(* Kommunikation mit der KL6581. *)
(* Communication with the KL6581. *)
fbKL6581(
	bInit			:= bInitCom,
	nIdx			:= 2,
	stKL6581_in		:= stKL6581_In,
	stKL6581_out	:= stKL6581_Out,
	bReady			=> ,
	bBusy			=> ,
	bError			=> ,
	iErrorID		=> ,
	str_KL6581		=> stKL6581);

GVL_AHDataModbus.EnOceanError	:= TO_UINT(fbKL6581.iErrorID);
(* Warten bis der Kommunikationsbaustein initialisiert wurde.*)
(* Wait until the communication function block has been initialized. *)
IF (NOT fbKL6581.bReady) THEN
	RETURN;
END_IF

FOR nSearchIdx:= 1 TO 8 DO
	arrEnOcean_Search[nSearchIdx](
		bStart:= TRUE, 
		str_KL6581:= stKL6581 , 
		byNode:= nSearchIdx, 
		bReceive=> , 
		iDevices=>arrDevices[nSearchIdx] , 
		ar_ID=> );
		
		MEMCPY(ADR(arrID[nSearchIdx,0]), ADR(arrEnOcean_Search[nSearchIdx].ar_ID), SIZEOF(arrEnOcean_Search[nSearchIdx].ar_ID)); 
END_FOR

//A_Gang_3_364()

A_Rum_2_351();
A_Rum_2_352();
A_Rum_2_353();
A_Rum_2_354();
A_Rum_2_355();
A_Rum_2_356();
A_Rum_2_357();
A_Rum_3_365();
A_Rum_3_361();
A_Rum_3_366();
A_Rum_3_367();
A_Rum_3_368();
A_Rum_3_369();
A_Rum_3_370();
//AtriumNiveau
A_AtriumNiveau();

ACTION A_AtriumNiveau:
fbAtriumNiveau_Tryk_PladeB(
	str_KL6581:=stKL6581 , 
	byNode:=0, 
	dw_ID:= 16#0029B92D, 
	str_EnOceanSwitch=> GVL_EnOcean.strEnOceanSwitch_AtriumNiveau_PladeB,
	by_Node=> , 
	bReceive=> );
(*
fbAtriumNiveau_Tryk_Sevice(
	str_KL6581:=stKL6581 , 
	byNode:=0, 
	dw_ID:= 16#00FEE4FE87, 
	str_EnOceanSwitch=> GVL_EnOcean.strEnOceanSwitch_AtriumNiveau_Service, 
	by_Node=> , 
	bReceive=> );
*)
END_ACTION

ACTION A_Rum_2_351:
fbRum_2_351_Tryk(
	str_KL6581:=stKL6581 , 
	byNode:=byNode_2 , 
	dw_ID:= 16#290EEB, 
	str_EnOceanSwitch=> GVL_EnOcean.strEnOceanSwitch_Rum_2_351, 
	by_Node=> , 
	bReceive=> );
END_ACTION

ACTION A_Rum_2_352:
fbRum_2_352_Tryk(
	str_KL6581:=stKL6581 , 
	byNode:=byNode_2 , 
	dw_ID:= 16#2F3276, 
	str_EnOceanSwitch=> GVL_EnOcean.strEnOceanSwitch_Rum_2_352, 
	by_Node=> , 
	bReceive=> );
END_ACTION

ACTION A_Rum_2_353:
fbRum_2_353_Tryk(
	str_KL6581:=stKL6581 , 
	byNode:=byNode_2 , 
	dw_ID:= 16#002E7C1F, 
	str_EnOceanSwitch=> GVL_EnOcean.strEnOceanSwitch_Rum_2_353, 
	by_Node=> , 
	bReceive=> );
END_ACTION

ACTION A_Rum_2_354:
fbRum_2_354_Tryk(
	str_KL6581:=stKL6581 , 
	byNode:=byNode_2 , 
	dw_ID:= 16#002F6627, 
	str_EnOceanSwitch=> GVL_EnOcean.strEnOceanSwitch_Rum_2_354, 
	by_Node=> , 
	bReceive=> );
END_ACTION

ACTION A_Rum_2_355:
fbRum_2_355_Tryk(
	str_KL6581:=stKL6581 , 
	byNode:=byNode_2 , 
	dw_ID:= 16#0029AD66, 
	str_EnOceanSwitch=> GVL_EnOcean.strEnOceanSwitch_Rum_2_355, 
	by_Node=> , 
	bReceive=> );
END_ACTION

ACTION A_Rum_2_356:
fbRum_2_356_Tryk(
	str_KL6581:=stKL6581 , 
	byNode:=byNode_2 , 
	dw_ID:= 16#0029AD36, 
	str_EnOceanSwitch=> GVL_EnOcean.strEnOceanSwitch_Rum_2_356, 
	by_Node=> , 
	bReceive=> );
END_ACTION

ACTION A_Rum_2_357:
fbRum_2_357_Tryk(
	str_KL6581:=stKL6581 , 
	byNode:=byNode_2 , 
	dw_ID:= 16#0029AD42, 
	str_EnOceanSwitch=> GVL_EnOcean.strEnOceanSwitch_Rum_2_357, 
	by_Node=> , 
	bReceive=> );
END_ACTION

ACTION A_Rum_3_361:
fbRum_3_361_Tryk_1(
	str_KL6581:=stKL6581 , 
	byNode:=byNode_2 , 
	dw_ID:= 16#29AD02, 
	str_EnOceanSwitch=> GVL_EnOcean.strEnOceanSwitch_Rum_3_361_1, 
	by_Node=> , 
	bReceive=> );


fbRum_3_361_Tryk_2(
	str_KL6581:=stKL6581 , 
	byNode:=byNode_2 , 
	dw_ID:= 16#0029ACFE, 
	str_EnOceanSwitch=> GVL_EnOcean.strEnOceanSwitch_Rum_3_361_2, 
	by_Node=> , 
	bReceive=> );
END_ACTION

ACTION A_Rum_3_365:
fbRum_3_365_Tryk(
	str_KL6581:=stKL6581 , 
	byNode:=byNode_2 , 
	dw_ID:= 16#0029AD2C, 
	str_EnOceanSwitch=> GVL_EnOcean.strEnOceanSwitch_Rum_3_365, 
	by_Node=> , 
	bReceive=> );
END_ACTION

ACTION A_Rum_3_366:
fbRum_3_366_Tryk(
	str_KL6581:=stKL6581 , 
	byNode:=byNode_2 , 
	dw_ID:= 16#0029AD33, 
	str_EnOceanSwitch=> GVL_EnOcean.strEnOceanSwitch_Rum_3_366, 
	by_Node=> , 
	bReceive=> );
END_ACTION

ACTION A_Rum_3_367:
fbRum_3_367_Tryk(
	str_KL6581:=stKL6581 , 
	byNode:=byNode_2 , 
	dw_ID:= 16#0029AD1B, 
	str_EnOceanSwitch=> GVL_EnOcean.strEnOceanSwitch_Rum_3_367, 
	by_Node=> , 
	bReceive=> );
END_ACTION

ACTION A_Rum_3_368:
fbRum_3_368_Tryk(
	str_KL6581:=stKL6581 , 
	byNode:=byNode_2 , 
	dw_ID:= 16#0029AD61, 
	str_EnOceanSwitch=> GVL_EnOcean.strEnOceanSwitch_Rum_3_368, 
	by_Node=> , 
	bReceive=> );
END_ACTION

ACTION A_Rum_3_369:
fbRum_3_369_Tryk(
	str_KL6581:=stKL6581 , 
	byNode:=byNode_2 , 
	dw_ID:= 16#0029AD37, 
	str_EnOceanSwitch=> GVL_EnOcean.strEnOceanSwitch_Rum_3_369, 
	by_Node=> , 
	bReceive=> );
END_ACTION

ACTION A_Rum_3_370:
fbRum_3_370_Tryk(
	str_KL6581:=stKL6581 , 
	byNode:=byNode_2 , 
	dw_ID:= 16#002F665E, 
	str_EnOceanSwitch=> GVL_EnOcean.strEnOceanSwitch_Rum_3_370, 
	by_Node=> , 
	bReceive=> );
END_ACTION

END_PROGRAM

// ---- POUs/MAIN.TcPOU
PROGRAM MAIN
VAR
	nAlive: INT;
	breset: BOOL;
	nDemoVariable : INT;
	nCX8200_State	AT %I*	: UINT;
END_VAR

VAR PERSISTENT
	nDemoVar_Persist: INT;
END_VAR

nAlive:= nAlive + 1;
GVL_AHDataModbus.nCX8200_State_MB := nCX8200_State;

P_SystemDK.M_nCyclic(bReset := breset );
P_DALI_DIAG();
//P_EnOcean(); Testing fast task
DALI_Commissioning();
P_DALI_Energy_Line();
P_AHModbusComm();
P_Foldedoer_3_366();

//Gange
P_Gang_2_350();
P_Gang_3_362A();
P_Gang_3_363A();
P_Gang_3_363B();
P_Gang_3_364();
P_gang_3_309();
//Rum
P_Rum_2_351();
P_Rum_2_352();
P_Rum_2_353();
P_Rum_2_354();
P_Rum_2_355();
P_Rum_2_356();
P_Rum_2_357();
P_Rum_3_361();
P_Rum_3_366();
P_Rum_3_367();
P_Rum_3_368();
P_Rum_3_369();
P_Rum_3_370();

//P_Lys_Grp0();
//P_DALI_Energy_Firmware_Test();
P_Trappe();

END_PROGRAM

// ---- POUs/Tester/P_Test_TypeA.TcPOU
PROGRAM P_Test_TypeA
VAR
	fbTA: FB_FunctionType_A;
	bButtonZone1 			: BOOL;
	bButtonZone2 			: BOOL;
	bPIR 					: BOOL;
	fLuxOn 					: REAL := 500;
	fLuxDim 				: REAL := 200;
	tPIRDim 				: TIME := T#15M;
	tPIROff 				: TIME := T#30M;
	
	//Output from FB
	fLuxZone1 				: REAL;
	bDimUp					: BOOL:= FALSE;
	bDimDwn 				: BOOL:= FALSE;
	bOnZone1 				: BOOL;
	bOffZone1 				: BOOL:= TRUE;
	bAutoZone1 				: BOOL:= TRUE;
	
	bAutoZone2 				: BOOL:= TRUE;
	bOnZone2 				: BOOL;
	bOffZone2 				: BOOL:= TRUE;
	
END_VAR


fbTA(
	bButtonZone1:= bButtonZone1, 
	bButtonZone2:= bButtonZone2 , 
	bPIR:= bPIR, 
	fLuxOn:= fLuxOn, 
	fLuxDim:= fLuxDim, 
	tPIRDim:= tPIRDim, 
	tPIROff:= tPIROff, 
	fLuxZone1=> fLuxZone1, 
	bDimUp=> bDimUp , 
	bDimDwn=> bDimDwn, 
	bOnZone1=> bOnZone1, 
	bOffZone1=> bOffZone1, 
	bAutoZone1=> bAutoZone1, 
	bAutoZone2=> bAutoZone2, 
	bOnZone2=> bOnZone2, 
	bOffZone2=> bOffZone2);

END_PROGRAM

// ---- GlobalTextList.TcGTLO
TEXTLIST GlobalTextList
  621 = '%d'
  6 = 'Bottom Button'
  482 = 'Button 1'
  720 = 'Button 2'
  1902 = 'DALI Line:'
  1180 = 'DI1 falling edge'
  1218 = 'DI1 rising edge'
  1726 = 'DI2 falling edge'
  1876 = 'DI2 rising edge'
  519 = 'Dim Dwn'
  63 = 'Dim Up'
  2135 = 'Do not lock process image in case of \nDALI commands from DI1 or DI2'
  967 = 'Gang 1.312A'
  256 = 'Gang 1.315'
  906 = 'Gang 1.316'
  207 = 'Gang 2.344'
  66 = 'Gang 2.344A'
  583 = 'Gang 2.350'
  985 = 'Gang 3.362A'
  67 = 'Gang 3.363A'
  173 = 'Gang 3.363B'
  406 = 'Gang 4.308'
  524 = 'Gang 6.310'
  316 = 'Gang 7.301'
  492 = 'Internal DALI power supply disabled'
  1771 = 'K-Bus Watchdog'
  1811 = 'Lockable bytes: changeable if "Offset 2" has the Value 85 (0x55).\nFor changing use decimal value.'
  43 = 'Lys Auto'
  444 = 'Lys Rum'
  489 = 'Lys Zone 1'
  2046 = 'Memory Bank:'
  23 = 'Name'
  926 = 'Name of byte in memory bank'
  22 = 'Offset'
  1329 = 'Offset in memory bank'
  708 = 'PIR'
  457 = 'PIR status'
  373 = 'Read'
  2418 = 'Reset inactive process image'
  874 = 'Rum 1.106'
  65 = 'Rum 1.108'
  175 = 'Rum 1.111A'
  924 = 'Rum 1.111C'
  219 = 'Rum 1.111D'
  690 = 'Rum 1.111E'
  912 = 'Rum 1.115'
  126 = 'Rum 1.118'
  215 = 'Rum 1.312A'
  725 = 'Rum 1.318'
  839 = 'Rum 1.319'
  456 = 'Rum 1.320'
  800 = 'Rum 1.321'
  622 = 'Rum 1.322'
  646 = 'Rum 1.323'
  966 = 'Rum 1.324'
  95 = 'Rum 1.325'
  335 = 'Rum 1.326'
  150 = 'Rum 1.327'
  651 = 'Rum 1.328'
  980 = 'Rum 1.330'
  262 = 'Rum 1115'
  642 = 'Rum 2.341'
  978 = 'Rum 2.345'
  736 = 'Rum 2.349'
  593 = 'Rum 2.351'
  122 = 'Rum 2.352'
  27 = 'Rum 2.353'
  41 = 'Rum 2.354'
  697 = 'Rum 2.355'
  826 = 'Rum 2.356'
  561 = 'Rum 2.357'
  415 = 'Rum 3.365'
  981 = 'Rum 3.366'
  865 = 'Rum 3.367'
  212 = 'Rum 3.368'
  921 = 'Rum 3.369'
  329 = 'Rum 3.370'
  430 = 'Rum 6.310 Sofagruppe'
  348 = 'Rum 6.327'
  891 = 'Rum 6.328'
  11 = 'Rum 6.329'
  72 = 'Rum 6.330B'
  197 = 'Rum 6.331'
  564 = 'Rum 6.333'
  997 = 'Rum 6.337'
  31 = 'Rum 6_330A'
  1041 = 'Short Address:'
  395 = 'SP_Lux: %.0f'
  525 = 'SP_Lux: %f'
  2458 = 'Terminal Event'
  849 = 'Test Type A'
  973 = 'Top Button'
  24 = 'Value Dec'
  1435 = 'Value decimal'
  25 = 'Value Hex'
  2231 = 'Value hexadecimal,\nto change use\nvalue decimal'
  374 = 'Write'
  1047 = 'Write default values'
  490 = 'Write parameters'
END_TEXTLIST

// ---- POUs/Alle_Rum/Gange/Gang_3_362A/Visualization_3_362A.TcVIS
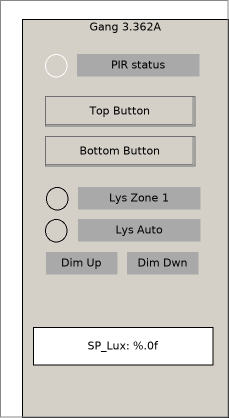
VISUALIZATION Visualization_3_362A  // 229x418
    RoundedRectangle (22,19 207x399), "Gang 3.362A"
    Rectangle (33,327 180x38), "SP_Lux: %.0f", text variable: P_Gang_3_362A.fbLys.fbLightCtrl.fLuxZone1
    Button (45,96 150x30), "Top Button"
        tap P_Gang_3_362A.bTopButtonZone1_Visu
    Button (45,136 150x30), "Bottom Button"
        tap P_Gang_3_362A.bBottomButtonZone1_Visu
    Ellipse (46,187 22x23), colour toggle: P_Gang_3_362A.fbLys.fbLightCtrl.bOnZone1
    Rectangle (78,187 122x22), "Lys Zone 1"
    Rectangle (46,252 71x22), "Dim Up", colour toggle: P_Gang_3_362A.fbLys.fbLightCtrl.bDimUp
    Rectangle (127,252 71x22), "Dim Dwn", colour toggle: P_Gang_3_362A.fbLys.fbLightCtrl.bDimDwn
    Ellipse (45,219 22x23), colour toggle: P_Gang_3_362A.fbLys.fbLightCtrl.bAutoZone1
    Rectangle (78,219 122x22), "Lys Auto"
    Ellipse (45,54 22x23), colour toggle: P_Gang_3_362A.fbLys.fbLightCtrl.bPIR
    Rectangle (77,54 122x22), "PIR status"
END_VISUALIZATION

// ---- POUs/Alle_Rum/Gange/Gang_3_363A/Visualization_3_363A.TcVIS
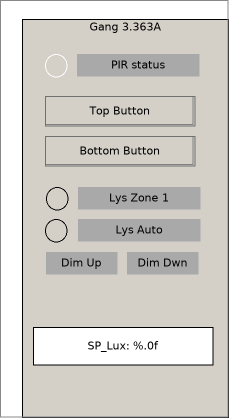
VISUALIZATION Visualization_3_363A  // 229x418
    RoundedRectangle (22,19 207x399), "Gang 3.363A"
    Rectangle (33,327 180x38), "SP_Lux: %.0f", text variable: P_Gang_3_363A.fbLys.fbLightCtrl.fLuxZone1
    Button (45,96 150x30), "Top Button"
        tap P_Gang_3_363A.bTopButtonZone1_Visu
    Button (45,136 150x30), "Bottom Button"
        tap P_Gang_3_363A.bBottomButtonZone1_Visu
    Ellipse (46,187 22x23), colour toggle: P_Gang_3_363A.fbLys.fbLightCtrl.bOnZone1
    Rectangle (78,187 122x22), "Lys Zone 1"
    Rectangle (46,252 71x22), "Dim Up", colour toggle: P_Gang_3_363A.fbLys.fbLightCtrl.bDimUp
    Rectangle (127,252 71x22), "Dim Dwn", colour toggle: P_Gang_3_363A.fbLys.fbLightCtrl.bDimDwn
    Ellipse (45,219 22x23), colour toggle: P_Gang_3_363A.fbLys.fbLightCtrl.bAutoZone1
    Rectangle (78,219 122x22), "Lys Auto"
    Ellipse (45,54 22x23), colour toggle: P_Gang_3_363A.fbLys.fbLightCtrl.bPIR
    Rectangle (77,54 122x22), "PIR status"
END_VISUALIZATION

// ---- POUs/Alle_Rum/Gange/Gang_3_363B/Visualization_3_363B.TcVIS
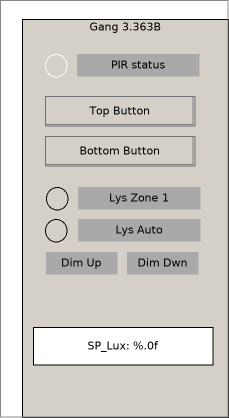
VISUALIZATION Visualization_3_363B  // 229x418
    RoundedRectangle (22,19 207x399), "Gang 3.363B"
    Rectangle (33,327 180x38), "SP_Lux: %.0f", text variable: P_Gang_3_362A.fbLys.fbLightCtrl.fLuxZone1
    Button (45,96 150x30), "Top Button"
        tap P_Gang_3_363B.bTopButtonZone1_Visu
    Button (45,136 150x30), "Bottom Button"
        tap P_Gang_3_363B.bBottomButtonZone1_Visu
    Ellipse (46,187 22x23), colour toggle: P_Gang_3_363B.fbLys.fbLightCtrl.bOnZone1
    Rectangle (78,187 122x22), "Lys Zone 1"
    Rectangle (46,252 71x22), "Dim Up", colour toggle: P_Gang_3_363B.fbLys.fbLightCtrl.bDimUp
    Rectangle (127,252 71x22), "Dim Dwn", colour toggle: P_Gang_3_363B.fbLys.fbLightCtrl.bDimDwn
    Ellipse (45,219 22x23), colour toggle: P_Gang_3_363B.fbLys.fbLightCtrl.bAutoZone1
    Rectangle (78,219 122x22), "Lys Auto"
    Ellipse (45,54 22x23), colour toggle: P_Gang_3_363B.fbLys.fbLightCtrl.bPIR
    Rectangle (77,54 122x22), "PIR status"
END_VISUALIZATION

// ---- POUs/Alle_Rum/Gange/Gang_3_364/Visualization_3_364.TcVIS
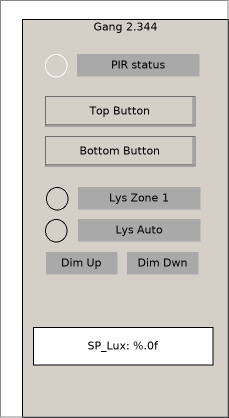
VISUALIZATION Visualization_3_364  // 229x418
    RoundedRectangle (22,19 207x399), "Gang 2.344"
    Rectangle (33,327 180x38), "SP_Lux: %.0f", text variable: P_Gang_3_364.fbLys.fbLightCtrl.fLuxZone1
    Button (45,96 150x30), "Top Button"
        tap P_Gang_3_364.bTopButtonZone1_Visu
    Button (45,136 150x30), "Bottom Button"
        tap P_Gang_3_364.bBottomButtonZone1_Visu
    Ellipse (46,187 22x23), colour toggle: P_Gang_3_364.fbLys.fbLightCtrl.bOnZone1
    Rectangle (78,187 122x22), "Lys Zone 1"
    Rectangle (46,252 71x22), "Dim Up", colour toggle: P_Gang_3_364.fbLys.fbLightCtrl.bDimUp
    Rectangle (127,252 71x22), "Dim Dwn", colour toggle: P_Gang_3_364.fbLys.fbLightCtrl.bDimDwn
    Ellipse (45,219 22x23), colour toggle: P_Gang_3_364.fbLys.fbLightCtrl.bAutoZone1
    Rectangle (78,219 122x22), "Lys Auto"
    Ellipse (45,54 22x23), colour toggle: P_Gang_3_364.fbLys.fbLightCtrl.bPIR
    Rectangle (77,54 122x22), "PIR status"
END_VISUALIZATION

// ---- POUs/Alle_Rum/Gange/Gang_2_350/Visualization_2_350.TcVIS
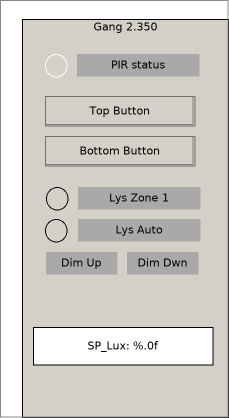
VISUALIZATION Visualization_2_350  // 229x418
    RoundedRectangle (22,19 207x399), "Gang 2.350"
    Rectangle (33,327 180x38), "SP_Lux: %.0f", text variable: P_Gang_3_364.fbLys.fbLightCtrl.fLuxZone1
    Button (45,96 150x30), "Top Button"
        tap P_Gang_2_350.bTopButtonZone1_Visu
    Button (45,136 150x30), "Bottom Button"
        tap P_Gang_2_350.bBottomButtonZone1_Visu
    Ellipse (46,187 22x23), colour toggle: P_Gang_2_350.fbLys.fbLightCtrl.bOnZone1
    Rectangle (78,187 122x22), "Lys Zone 1"
    Rectangle (46,252 71x22), "Dim Up", colour toggle: P_Gang_2_350.fbLys.fbLightCtrl.bDimUp
    Rectangle (127,252 71x22), "Dim Dwn", colour toggle: P_Gang_2_350.fbLys.fbLightCtrl.bDimDwn
    Ellipse (45,219 22x23), colour toggle: P_Gang_2_350.fbLys.fbLightCtrl.bAutoZone1
    Rectangle (78,219 122x22), "Lys Auto"
    Ellipse (45,54 22x23), colour toggle: P_Gang_2_350.fbLys.fbLightCtrl.bPIR
    Rectangle (77,54 122x22), "PIR status"
END_VISUALIZATION

// ---- POUs/Alle_Rum/Rum_Med_DALI_Pir/Rum_2_351/Visualization_2_351.TcVIS
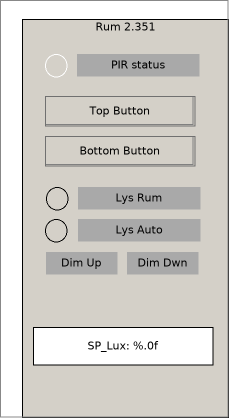
VISUALIZATION Visualization_2_351  // 229x418
    RoundedRectangle (22,19 207x399), "Rum 2.351"
    Rectangle (33,327 180x38), "SP_Lux: %.0f", text variable: P_Rum_2_351.fbLys.fbLightCtrl.fLuxZone1
    Button (45,96 150x30), "Top Button"
        tap P_Rum_2_351.bTopButtonZone1_Visu
    Button (45,136 150x30), "Bottom Button"
        tap P_Rum_2_351.bBottomButtonZone1_Visu
    Ellipse (46,187 22x23), colour toggle: P_Rum_2_351.fbLys.fbLightCtrl.bOnZone1
    Rectangle (78,187 122x22), "Lys Rum"
    Rectangle (46,252 71x22), "Dim Up", colour toggle: P_Rum_2_351.fbLys.fbLightCtrl.bDimUp
    Rectangle (127,252 71x22), "Dim Dwn", colour toggle: P_Rum_2_351.fbLys.fbLightCtrl.bDimDwn
    Ellipse (45,219 22x23), colour toggle: P_Rum_2_351.fbLys.fbLightCtrl.bAutoZone1
    Rectangle (78,219 122x22), "Lys Auto"
    Ellipse (45,54 22x23), colour toggle: P_Rum_2_351.fbLys.fbLightCtrl.bPIR
    Rectangle (77,54 122x22), "PIR status"
END_VISUALIZATION

// ---- POUs/Alle_Rum/Rum_Med_DALI_Pir/Rum_2_352/Visualization_2_352.TcVIS
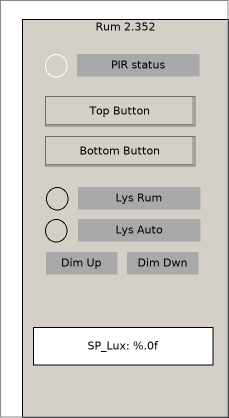
VISUALIZATION Visualization_2_352  // 229x418
    RoundedRectangle (22,19 207x399), "Rum 2.352"
    Rectangle (33,327 180x38), "SP_Lux: %.0f", text variable: P_Rum_2_351.fbLys.fbLightCtrl.fLuxZone1
    Button (45,96 150x30), "Top Button"
        tap P_Rum_2_352.bTopButtonZone1_Visu
    Button (45,136 150x30), "Bottom Button"
        tap P_Rum_2_352.bBottomButtonZone1_Visu
    Ellipse (46,187 22x23), colour toggle: P_Rum_2_352.fbLys.fbLightCtrl.bOnZone1
    Rectangle (78,187 122x22), "Lys Rum"
    Rectangle (46,252 71x22), "Dim Up", colour toggle: P_Rum_2_352.fbLys.fbLightCtrl.bDimUp
    Rectangle (127,252 71x22), "Dim Dwn", colour toggle: P_Rum_2_352.fbLys.fbLightCtrl.bDimDwn
    Ellipse (45,219 22x23), colour toggle: P_Rum_2_352.fbLys.fbLightCtrl.bAutoZone1
    Rectangle (78,219 122x22), "Lys Auto"
    Ellipse (45,54 22x23), colour toggle: P_Rum_2_352.fbLys.fbLightCtrl.bPIR
    Rectangle (77,54 122x22), "PIR status"
END_VISUALIZATION

// ---- POUs/Alle_Rum/Rum_Med_DALI_Pir/Rum_2_353/Visualization_2_353.TcVIS
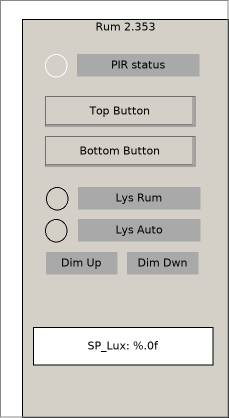
VISUALIZATION Visualization_2_353  // 229x418
    RoundedRectangle (22,19 207x399), "Rum 2.353"
    Rectangle (33,327 180x38), "SP_Lux: %.0f", text variable: P_Rum_2_353.fbLys.fbLightCtrl.fLuxZone1
    Button (45,96 150x30), "Top Button"
        tap P_Rum_2_353.bTopButtonZone1_Visu
    Button (45,136 150x30), "Bottom Button"
        tap P_Rum_2_353.bBottomButtonZone1_Visu
    Ellipse (46,187 22x23), colour toggle: P_Rum_2_353.fbLys.fbLightCtrl.bOnZone1
    Rectangle (78,187 122x22), "Lys Rum"
    Rectangle (46,252 71x22), "Dim Up", colour toggle: P_Rum_2_353.fbLys.fbLightCtrl.bDimUp
    Rectangle (127,252 71x22), "Dim Dwn", colour toggle: P_Rum_2_353.fbLys.fbLightCtrl.bDimDwn
    Ellipse (45,219 22x23), colour toggle: P_Rum_2_353.fbLys.fbLightCtrl.bAutoZone1
    Rectangle (78,219 122x22), "Lys Auto"
    Ellipse (45,54 22x23), colour toggle: P_Rum_2_353.fbLys.fbLightCtrl.bPIR
    Rectangle (77,54 122x22), "PIR status"
END_VISUALIZATION

// ---- POUs/Alle_Rum/Rum_Med_DALI_Pir/Rum_2_354/Visualization_2_354.TcVIS
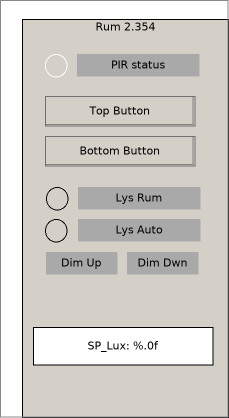
VISUALIZATION Visualization_2_354  // 229x418
    RoundedRectangle (22,19 207x399), "Rum 2.354"
    Rectangle (33,327 180x38), "SP_Lux: %.0f", text variable: P_Rum_2_354.fbLys.fbLightCtrl.fLuxZone1
    Button (45,96 150x30), "Top Button"
        tap P_Rum_2_354.bTopButtonZone1_Visu
    Button (45,136 150x30), "Bottom Button"
        tap P_Rum_2_354.bBottomButtonZone1_Visu
    Ellipse (46,187 22x23), colour toggle: P_Rum_2_354.fbLys.fbLightCtrl.bOnZone1
    Rectangle (78,187 122x22), "Lys Rum"
    Rectangle (46,252 71x22), "Dim Up", colour toggle: P_Rum_2_354.fbLys.fbLightCtrl.bDimUp
    Rectangle (127,252 71x22), "Dim Dwn", colour toggle: P_Rum_2_354.fbLys.fbLightCtrl.bDimDwn
    Ellipse (45,219 22x23), colour toggle: P_Rum_2_354.fbLys.fbLightCtrl.bAutoZone1
    Rectangle (78,219 122x22), "Lys Auto"
    Ellipse (45,54 22x23), colour toggle: P_Rum_2_354.fbLys.fbLightCtrl.bPIR
    Rectangle (77,54 122x22), "PIR status"
END_VISUALIZATION

// ---- POUs/Alle_Rum/Rum_Med_DALI_Pir/Rum_2_357/Visualization_2_357.TcVIS
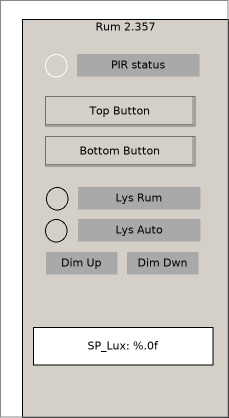
VISUALIZATION Visualization_2_357  // 229x418
    RoundedRectangle (22,19 207x399), "Rum 2.357"
    Rectangle (33,327 180x38), "SP_Lux: %.0f", text variable: P_Rum_2_357.fbLys.fbLightCtrl.fLuxZone1
    Button (45,96 150x30), "Top Button"
        tap P_Rum_2_357.bTopButtonZone1_Visu
    Button (45,136 150x30), "Bottom Button"
        tap P_Rum_2_357.bBottomButtonZone1_Visu
    Ellipse (46,187 22x23), colour toggle: P_Rum_2_357.fbLys.fbLightCtrl.bOnZone1
    Rectangle (78,187 122x22), "Lys Rum"
    Rectangle (46,252 71x22), "Dim Up", colour toggle: P_Rum_2_357.fbLys.fbLightCtrl.bDimUp
    Rectangle (127,252 71x22), "Dim Dwn", colour toggle: P_Rum_2_357.fbLys.fbLightCtrl.bDimDwn
    Ellipse (45,219 22x23), colour toggle: P_Rum_2_357.fbLys.fbLightCtrl.bAutoZone1
    Rectangle (78,219 122x22), "Lys Auto"
    Ellipse (45,54 22x23), colour toggle: P_Rum_2_357.fbLys.fbLightCtrl.bPIR
    Rectangle (77,54 122x22), "PIR status"
END_VISUALIZATION

// ---- POUs/Alle_Rum/Rum_Med_DALI_Pir/Rum_2_355/Visualization_2_355.TcVIS
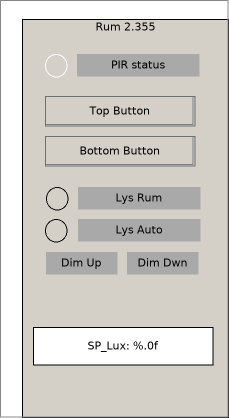
VISUALIZATION Visualization_2_355  // 229x418
    RoundedRectangle (22,19 207x399), "Rum 2.355"
    Rectangle (33,327 180x38), "SP_Lux: %.0f", text variable: P_Rum_2_355.fbLys.fbLightCtrl.fLuxZone1
    Button (45,96 150x30), "Top Button"
        tap P_Rum_2_355.bTopButtonZone1_Visu
    Button (45,136 150x30), "Bottom Button"
        tap P_Rum_2_355.bBottomButtonZone1_Visu
    Ellipse (46,187 22x23), colour toggle: P_Rum_2_355.fbLys.fbLightCtrl.bOnZone1
    Rectangle (78,187 122x22), "Lys Rum"
    Rectangle (46,252 71x22), "Dim Up", colour toggle: P_Rum_2_355.fbLys.fbLightCtrl.bDimUp
    Rectangle (127,252 71x22), "Dim Dwn", colour toggle: P_Rum_2_355.fbLys.fbLightCtrl.bDimDwn
    Ellipse (45,219 22x23), colour toggle: P_Rum_2_355.fbLys.fbLightCtrl.bAutoZone1
    Rectangle (78,219 122x22), "Lys Auto"
    Ellipse (45,54 22x23), colour toggle: P_Rum_2_355.fbLys.fbLightCtrl.bPIR
    Rectangle (77,54 122x22), "PIR status"
END_VISUALIZATION

// ---- POUs/Alle_Rum/Rum_Med_DALI_Pir/Rum_2_356/Visualization_2_356.TcVIS
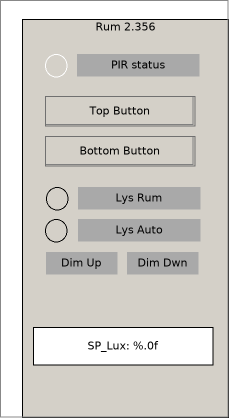
VISUALIZATION Visualization_2_356  // 229x418
    RoundedRectangle (22,19 207x399), "Rum 2.356"
    Rectangle (33,327 180x38), "SP_Lux: %.0f", text variable: P_Rum_2_356.fbLys.fbLightCtrl.fLuxZone1
    Button (45,96 150x30), "Top Button"
        tap P_Rum_2_356.bTopButtonZone1_Visu
    Button (45,136 150x30), "Bottom Button"
        tap P_Rum_2_356.bBottomButtonZone1_Visu
    Ellipse (46,187 22x23), colour toggle: P_Rum_2_356.fbLys.fbLightCtrl.bOnZone1
    Rectangle (78,187 122x22), "Lys Rum"
    Rectangle (46,252 71x22), "Dim Up", colour toggle: P_Rum_2_356.fbLys.fbLightCtrl.bDimUp
    Rectangle (127,252 71x22), "Dim Dwn", colour toggle: P_Rum_2_356.fbLys.fbLightCtrl.bDimDwn
    Ellipse (45,219 22x23), colour toggle: P_Rum_2_356.fbLys.fbLightCtrl.bAutoZone1
    Rectangle (78,219 122x22), "Lys Auto"
    Ellipse (45,54 22x23), colour toggle: P_Rum_2_356.fbLys.fbLightCtrl.bPIR
    Rectangle (77,54 122x22), "PIR status"
END_VISUALIZATION

// ---- POUs/Alle_Rum/Rum_Med_DALI_Pir/Rum_3_361/Visualization_2_357_1.TcVIS
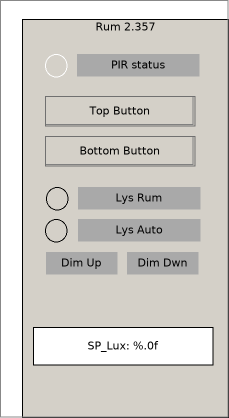
VISUALIZATION Visualization_2_357_1  // 229x418
    RoundedRectangle (22,19 207x399), "Rum 2.357"
    Rectangle (33,327 180x38), "SP_Lux: %.0f", text variable: P_Rum_2_357.fbLys.fbLightCtrl.fLuxZone1
    Button (45,96 150x30), "Top Button"
        tap P_Rum_2_357.bTopButtonZone1_Visu
    Button (45,136 150x30), "Bottom Button"
        tap P_Rum_2_357.bBottomButtonZone1_Visu
    Ellipse (46,187 22x23), colour toggle: P_Rum_2_357.fbLys.fbLightCtrl.bOnZone1
    Rectangle (78,187 122x22), "Lys Rum"
    Rectangle (46,252 71x22), "Dim Up", colour toggle: P_Rum_2_357.fbLys.fbLightCtrl.bDimUp
    Rectangle (127,252 71x22), "Dim Dwn", colour toggle: P_Rum_2_357.fbLys.fbLightCtrl.bDimDwn
    Ellipse (45,219 22x23), colour toggle: P_Rum_2_357.fbLys.fbLightCtrl.bAutoZone1
    Rectangle (78,219 122x22), "Lys Auto"
    Ellipse (45,54 22x23), colour toggle: P_Rum_2_357.fbLys.fbLightCtrl.bPIR
    Rectangle (77,54 122x22), "PIR status"
END_VISUALIZATION

// ---- POUs/Alle_Rum/Rum_Med_DALI_Pir/Rum_3_365/Visualization_3_365.TcVIS
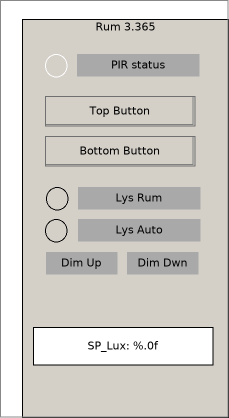
VISUALIZATION Visualization_3_365  // 229x418
    RoundedRectangle (22,19 207x399), "Rum 3.365"
    Rectangle (33,327 180x38), "SP_Lux: %.0f", text variable: P_Rum_3_365.fbLys.fbLightCtrl.fLuxZone1
    Button (45,96 150x30), "Top Button"
        tap P_Rum_3_365.bTopButtonZone1_Visu
    Button (45,136 150x30), "Bottom Button"
        tap P_Rum_3_365.bBottomButtonZone1_Visu
    Ellipse (46,187 22x23), colour toggle: P_Rum_3_365.fbLys.fbLightCtrl.bOnZone1
    Rectangle (78,187 122x22), "Lys Rum"
    Rectangle (46,252 71x22), "Dim Up", colour toggle: P_Rum_3_365.fbLys.fbLightCtrl.bDimUp
    Rectangle (127,252 71x22), "Dim Dwn", colour toggle: P_Rum_3_365.fbLys.fbLightCtrl.bDimDwn
    Ellipse (45,219 22x23), colour toggle: P_Rum_3_365.fbLys.fbLightCtrl.bAutoZone1
    Rectangle (78,219 122x22), "Lys Auto"
    Ellipse (45,54 22x23), colour toggle: P_Rum_3_365.fbLys.fbLightCtrl.bPIR
    Rectangle (77,54 122x22), "PIR status"
END_VISUALIZATION

// ---- POUs/Alle_Rum/Rum_Med_DALI_Pir/Rum_3_367/Visualization_3_367.TcVIS
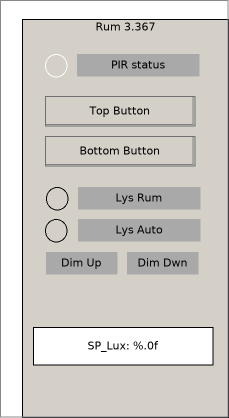
VISUALIZATION Visualization_3_367  // 229x418
    RoundedRectangle (22,19 207x399), "Rum 3.367"
    Rectangle (33,327 180x38), "SP_Lux: %.0f", text variable: P_Rum_3_367.fbLys.fbLightCtrl.fLuxZone1
    Button (45,96 150x30), "Top Button"
        tap P_Rum_3_367.bTopButtonZone1_Visu
    Button (45,136 150x30), "Bottom Button"
        tap P_Rum_3_367.bBottomButtonZone1_Visu
    Ellipse (46,187 22x23), colour toggle: P_Rum_3_367.fbLys.fbLightCtrl.bOnZone1
    Rectangle (78,187 122x22), "Lys Rum"
    Rectangle (46,252 71x22), "Dim Up", colour toggle: P_Rum_3_367.fbLys.fbLightCtrl.bDimUp
    Rectangle (127,252 71x22), "Dim Dwn", colour toggle: P_Rum_3_367.fbLys.fbLightCtrl.bDimDwn
    Ellipse (45,219 22x23), colour toggle: P_Rum_3_367.fbLys.fbLightCtrl.bAutoZone1
    Rectangle (78,219 122x22), "Lys Auto"
    Ellipse (45,54 22x23), colour toggle: P_Rum_3_367.fbLys.fbLightCtrl.bPIR
    Rectangle (77,54 122x22), "PIR status"
END_VISUALIZATION

// ---- POUs/Alle_Rum/Rum_Med_DALI_Pir/Rum_3_369/Visualization_3_369.TcVIS
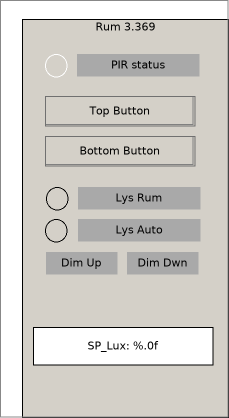
VISUALIZATION Visualization_3_369  // 229x418
    RoundedRectangle (22,19 207x399), "Rum 3.369"
    Rectangle (33,327 180x38), "SP_Lux: %.0f", text variable: P_Rum_3_369.fbLys.fbLightCtrl.fLuxZone1
    Button (45,96 150x30), "Top Button"
        tap P_Rum_3_369.bTopButtonZone1_Visu
    Button (45,136 150x30), "Bottom Button"
        tap P_Rum_3_369.bBottomButtonZone1_Visu
    Ellipse (46,187 22x23), colour toggle: P_Rum_3_369.fbLys.fbLightCtrl.bOnZone1
    Rectangle (78,187 122x22), "Lys Rum"
    Rectangle (46,252 71x22), "Dim Up", colour toggle: P_Rum_3_369.fbLys.fbLightCtrl.bDimUp
    Rectangle (127,252 71x22), "Dim Dwn", colour toggle: P_Rum_3_369.fbLys.fbLightCtrl.bDimDwn
    Ellipse (45,219 22x23), colour toggle: P_Rum_3_369.fbLys.fbLightCtrl.bAutoZone1
    Rectangle (78,219 122x22), "Lys Auto"
    Ellipse (45,54 22x23), colour toggle: P_Rum_3_369.fbLys.fbLightCtrl.bPIR
    Rectangle (77,54 122x22), "PIR status"
END_VISUALIZATION

// ---- POUs/Alle_Rum/Rum_Med_DALI_Pir/Rum_3_370/Visualization_3_370.TcVIS
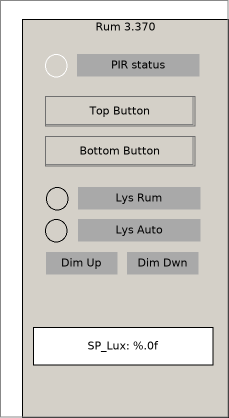
VISUALIZATION Visualization_3_370  // 229x418
    RoundedRectangle (22,19 207x399), "Rum 3.370"
    Rectangle (33,327 180x38), "SP_Lux: %.0f", text variable: P_Rum_3_370.fbLys.fbLightCtrl.fLuxZone1
    Button (45,96 150x30), "Top Button"
        tap P_Rum_3_370.bTopButtonZone1_Visu
    Button (45,136 150x30), "Bottom Button"
        tap P_Rum_3_370.bBottomButtonZone1_Visu
    Ellipse (46,187 22x23), colour toggle: P_Rum_3_370.fbLys.fbLightCtrl.bOnZone1
    Rectangle (78,187 122x22), "Lys Rum"
    Rectangle (46,252 71x22), "Dim Up", colour toggle: P_Rum_3_370.fbLys.fbLightCtrl.bDimUp
    Rectangle (127,252 71x22), "Dim Dwn", colour toggle: P_Rum_3_370.fbLys.fbLightCtrl.bDimDwn
    Ellipse (45,219 22x23), colour toggle: P_Rum_3_370.fbLys.fbLightCtrl.bAutoZone1
    Rectangle (78,219 122x22), "Lys Auto"
    Ellipse (45,54 22x23), colour toggle: P_Rum_3_370.fbLys.fbLightCtrl.bPIR
    Rectangle (77,54 122x22), "PIR status"
END_VISUALIZATION

// ---- POUs/DALI/DALI_Setup/VISUs/TextLists/TextList_Dialogs.TcTLO
TEXTLIST TextList_Dialogs
  0 = 'Select the function'
  1 = 'Control Gears - Commands'
  2 = 'Control Gears - Addressing'
  3 = 'Control Gears - Parameters'
  4 = 'Control Gears - Groups'
  5 = 'Control Gears - Scenes'
  6 = 'Control Gears - Memory Pages'
  7 = 'Control Gears - Set Fading'
  8 = 'Control Gears - Device Type 1 (Emergency lighting)'
  9 = 'Control Gears - Device Type 4 (Incandescent lamp)'
  10 = 'Control Gears - Device Type 6 (LED)'
  11 = 'Control Gears - Device Type 7 (Switching)'
  12 = 'Control Devices - Addressing'
  13 = 'Control Devices - Parameters'
  15 = 'Control Devices - Device Type 1 (Push button)'
  16 = 'Control Devices - Device Type 2 (Absolute input)'
  17 = 'Control Devices - Device Type 3 (Occupancy sensor)'
  18 = 'Control Devices - Device Type 4 (Light sensor)'
  19 = 'Control Devices - Device Type 0 (Generic instance)'
  20 = 'Control Devices - Memory Pages'
  14 = 'Control Devices - Identify'
   = ''
END_TEXTLIST

// ---- POUs/DALI/DALI_Setup/VISUs/Visu_DALICommissioning/Visu_Part102Addressing.TcVIS
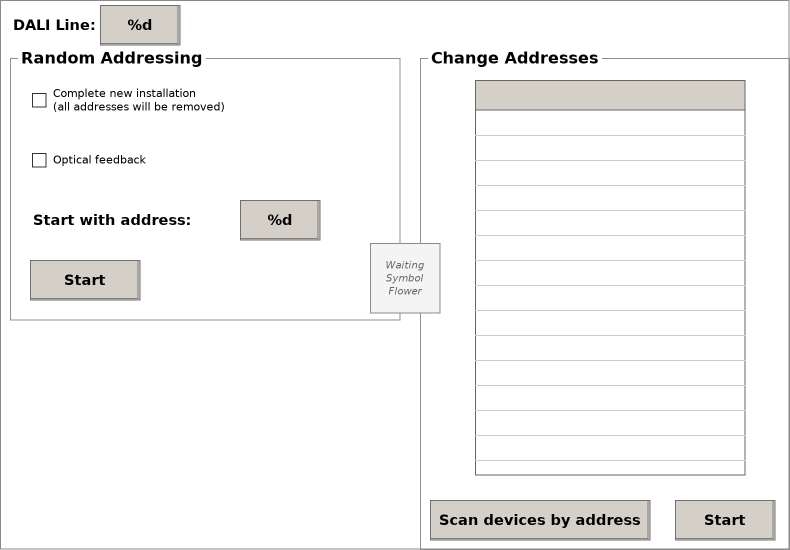
VISUALIZATION Visu_Part102Addressing  // 790x550
    GroupBox (420,50 370x500), "Change Addresses"
        Table (55,30 270x395), data array: DALI_Commissioning.fbPart102Addressing.aChangeAddressList
            p3854506369: DALI_Commissioning.fbPart102Addressing.aChangeAddressList[INDEX].nOldAddress
            p1892666644: DALI_Commissioning.fbPart102Addressing.aChangeAddressList[INDEX].nNewAddress
            p338671338: DALI_Commissioning.fbPart102Addressing.aChangeAddressList[INDEX].nRandomAddress
            p2170511999: DALI_Commissioning.fbPart102Addressing.aChangeAddressList[INDEX].nErrors
            Columns.Column.[0].Template: DALI_Commissioning.fbPart102Addressing.aNoShortAddress[INDEX]
            Columns.Column.[1].Template: DALI_Commissioning.fbPart102Addressing.aNoShortAddress[INDEX]; OnMouseClick: write the text variable via Default, min 0, max 63, title "New Short Address"
        Button (255,450 100x40), "Start"
            OnMouseClick: execute { DALI_Commissioning.fbPart102Addressing.bStartChangeAddress := TRUE; }
        Button (10,450 220x40), "Scan devices by address"
            OnMouseClick: execute { DALI_Commissioning.fbPart102Addressing.bScanDevices := TRUE; }
    GroupBox (10,50 390x270), "Random Addressing"
        Button (20,210 110x40), "Start"
            OnMouseClick: execute { DALI_Commissioning.fbPart102Addressing.bStartRandomAddressing := TRUE; }
        Checkbox (20,30 360x40), "Complete new installation (all addresses will be removed)", variable: DALI_Commissioning.fbPart102Addressing.bNewInstallation
        Checkbox (20,90 360x40), "Optical feedback", variable: DALI_Commissioning.fbPart102Addressing.bOpticalFeedback
        Textfield (20,150 200x40), "Start with address:"
        Button (230,150 80x40), "%d", text variable: DALI_Commissioning.fbPart102Addressing.nStartAddress
            OnMouseClick: write the text variable via Default, min 0, max 63, title "Insert Short Address"
    WaitingSymbolFlower (370,243 70x70), invisible if: DALI_Commissioning.fbPart102Addressing.bHideWaitSymbol
    Group (10,5 170x40)
        Textfield (0,0 110x40), "DALI Line:"
        Button (90,0 80x40), "%d", text variable: GVL_Internal.nDALILine
            OnMouseClick: write the text variable via Default, min 1, max 10, title "Choose line"
END_VISUALIZATION

// ---- POUs/DALI/DALI_Setup/VISUs/Visu_DALICommissioning/Visu_Part102Groups.TcVIS
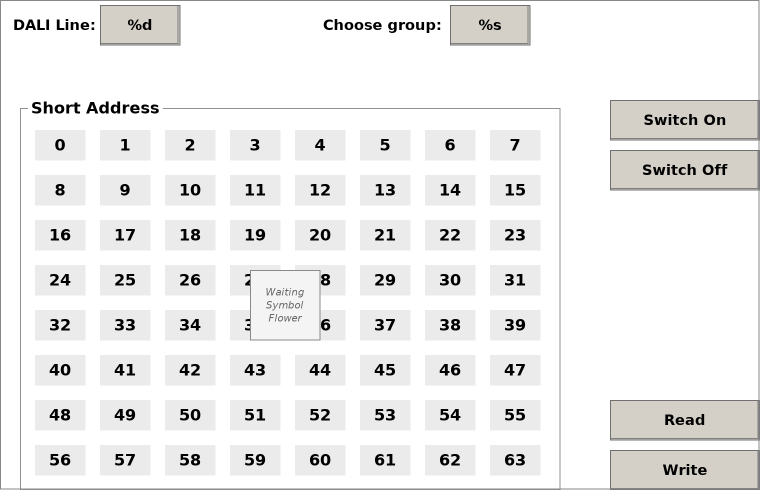
VISUALIZATION Visu_Part102Groups  // 760x490
    GroupBox (20,100 540x390), "Short Address"
        Textfield (15,30 50x30), "0", colour toggle: DALI_Commissioning.fbPart102Groups.aShowAlarmState[0] = TRUE, invisible if: DALI_Commissioning.fbPart102Groups.aActivateButton[0] = FALSE, input disabled if: DALI_Commissioning.fbPart102Groups.aActivateButton[0] = FALSE
            OnMouseClick: execute { DALI_Commissioning.fbPart102Groups.aButtonClick[0] := TRUE; }
        Textfield (80,30 50x30), "1", colour toggle: DALI_Commissioning.fbPart102Groups.aShowAlarmState[1] = TRUE, invisible if: DALI_Commissioning.fbPart102Groups.aActivateButton[1] = FALSE, input disabled if: DALI_Commissioning.fbPart102Groups.aActivateButton[1] = FALSE
            OnMouseClick: execute { DALI_Commissioning.fbPart102Groups.aButtonClick[1] := TRUE; }
        Textfield (145,30 50x30), "2", colour toggle: DALI_Commissioning.fbPart102Groups.aShowAlarmState[2] = TRUE, invisible if: DALI_Commissioning.fbPart102Groups.aActivateButton[2] = FALSE, input disabled if: DALI_Commissioning.fbPart102Groups.aActivateButton[2] = FALSE
            OnMouseClick: execute { DALI_Commissioning.fbPart102Groups.aButtonClick[2] := TRUE; }
        Textfield (210,30 50x30), "3", colour toggle: DALI_Commissioning.fbPart102Groups.aShowAlarmState[3] = TRUE, invisible if: DALI_Commissioning.fbPart102Groups.aActivateButton[3] = FALSE, input disabled if: DALI_Commissioning.fbPart102Groups.aActivateButton[3] = FALSE
            OnMouseClick: execute { DALI_Commissioning.fbPart102Groups.aButtonClick[3] := TRUE; }
        Textfield (275,30 50x30), "4", colour toggle: DALI_Commissioning.fbPart102Groups.aShowAlarmState[4] = TRUE, invisible if: DALI_Commissioning.fbPart102Groups.aActivateButton[4] = FALSE, input disabled if: DALI_Commissioning.fbPart102Groups.aActivateButton[4] = FALSE
            OnMouseClick: execute { DALI_Commissioning.fbPart102Groups.aButtonClick[4] := TRUE; }
        Textfield (340,30 50x30), "5", colour toggle: DALI_Commissioning.fbPart102Groups.aShowAlarmState[5] = TRUE, invisible if: DALI_Commissioning.fbPart102Groups.aActivateButton[5] = FALSE, input disabled if: DALI_Commissioning.fbPart102Groups.aActivateButton[5] = FALSE
            OnMouseClick: execute { DALI_Commissioning.fbPart102Groups.aButtonClick[5] := TRUE; }
        Textfield (405,30 50x30), "6", colour toggle: DALI_Commissioning.fbPart102Groups.aShowAlarmState[6] = TRUE, invisible if: DALI_Commissioning.fbPart102Groups.aActivateButton[6] = FALSE, input disabled if: DALI_Commissioning.fbPart102Groups.aActivateButton[6] = FALSE
            OnMouseClick: execute { DALI_Commissioning.fbPart102Groups.aButtonClick[6] := TRUE; }
        Textfield (470,30 50x30), "7", colour toggle: DALI_Commissioning.fbPart102Groups.aShowAlarmState[7] = TRUE, invisible if: DALI_Commissioning.fbPart102Groups.aActivateButton[7] = FALSE, input disabled if: DALI_Commissioning.fbPart102Groups.aActivateButton[7] = FALSE
            OnMouseClick: execute { DALI_Commissioning.fbPart102Groups.aButtonClick[7] := TRUE; }
        Textfield (15,75 50x30), "8", colour toggle: DALI_Commissioning.fbPart102Groups.aShowAlarmState[8] = TRUE, invisible if: DALI_Commissioning.fbPart102Groups.aActivateButton[8] = FALSE, input disabled if: DALI_Commissioning.fbPart102Groups.aActivateButton[8] = FALSE
            OnMouseClick: execute { DALI_Commissioning.fbPart102Groups.aButtonClick[8] := TRUE; }
        Textfield (80,75 50x30), "9", colour toggle: DALI_Commissioning.fbPart102Groups.aShowAlarmState[9] = TRUE, invisible if: DALI_Commissioning.fbPart102Groups.aActivateButton[9] = FALSE, input disabled if: DALI_Commissioning.fbPart102Groups.aActivateButton[9] = FALSE
            OnMouseClick: execute { DALI_Commissioning.fbPart102Groups.aButtonClick[9] := TRUE; }
        Textfield (145,75 50x30), "10", colour toggle: DALI_Commissioning.fbPart102Groups.aShowAlarmState[10] = TRUE, invisible if: DALI_Commissioning.fbPart102Groups.aActivateButton[10] = FALSE, input disabled if: DALI_Commissioning.fbPart102Groups.aActivateButton[10] = FALSE
            OnMouseClick: execute { DALI_Commissioning.fbPart102Groups.aButtonClick[10] := TRUE; }
        Textfield (210,75 50x30), "11", colour toggle: DALI_Commissioning.fbPart102Groups.aShowAlarmState[11] = TRUE, invisible if: DALI_Commissioning.fbPart102Groups.aActivateButton[11] = FALSE, input disabled if: DALI_Commissioning.fbPart102Groups.aActivateButton[11] = FALSE
            OnMouseClick: execute { DALI_Commissioning.fbPart102Groups.aButtonClick[11] := TRUE; }
        Textfield (275,75 50x30), "12", colour toggle: DALI_Commissioning.fbPart102Groups.aShowAlarmState[12] = TRUE, invisible if: DALI_Commissioning.fbPart102Groups.aActivateButton[12] = FALSE, input disabled if: DALI_Commissioning.fbPart102Groups.aActivateButton[12] = FALSE
            OnMouseClick: execute { DALI_Commissioning.fbPart102Groups.aButtonClick[12] := TRUE; }
        Textfield (340,75 50x30), "13", colour toggle: DALI_Commissioning.fbPart102Groups.aShowAlarmState[13] = TRUE, invisible if: DALI_Commissioning.fbPart102Groups.aActivateButton[13] = FALSE, input disabled if: DALI_Commissioning.fbPart102Groups.aActivateButton[13] = FALSE
            OnMouseClick: execute { DALI_Commissioning.fbPart102Groups.aButtonClick[13] := TRUE; }
        Textfield (405,75 50x30), "14", colour toggle: DALI_Commissioning.fbPart102Groups.aShowAlarmState[14] = TRUE, invisible if: DALI_Commissioning.fbPart102Groups.aActivateButton[14] = FALSE, input disabled if: DALI_Commissioning.fbPart102Groups.aActivateButton[14] = FALSE
            OnMouseClick: execute { DALI_Commissioning.fbPart102Groups.aButtonClick[14] := TRUE; }
        Textfield (470,75 50x30), "15", colour toggle: DALI_Commissioning.fbPart102Groups.aShowAlarmState[15] = TRUE, invisible if: DALI_Commissioning.fbPart102Groups.aActivateButton[15] = FALSE, input disabled if: DALI_Commissioning.fbPart102Groups.aActivateButton[15] = FALSE
            OnMouseClick: execute { DALI_Commissioning.fbPart102Groups.aButtonClick[15] := TRUE; }
        Textfield (15,120 50x30), "16", colour toggle: DALI_Commissioning.fbPart102Groups.aShowAlarmState[16] = TRUE, invisible if: DALI_Commissioning.fbPart102Groups.aActivateButton[16] = FALSE, input disabled if: DALI_Commissioning.fbPart102Groups.aActivateButton[16] = FALSE
            OnMouseClick: execute { DALI_Commissioning.fbPart102Groups.aButtonClick[16] := TRUE; }
        Textfield (80,120 50x30), "17", colour toggle: DALI_Commissioning.fbPart102Groups.aShowAlarmState[17] = TRUE, invisible if: DALI_Commissioning.fbPart102Groups.aActivateButton[17] = FALSE, input disabled if: DALI_Commissioning.fbPart102Groups.aActivateButton[17] = FALSE
            OnMouseClick: execute { DALI_Commissioning.fbPart102Groups.aButtonClick[17] := TRUE; }
        Textfield (145,120 50x30), "18", colour toggle: DALI_Commissioning.fbPart102Groups.aShowAlarmState[18] = TRUE, invisible if: DALI_Commissioning.fbPart102Groups.aActivateButton[18] = FALSE, input disabled if: DALI_Commissioning.fbPart102Groups.aActivateButton[18] = FALSE
            OnMouseClick: execute { DALI_Commissioning.fbPart102Groups.aButtonClick[18] := TRUE; }
        Textfield (210,120 50x30), "19", colour toggle: DALI_Commissioning.fbPart102Groups.aShowAlarmState[19] = TRUE, invisible if: DALI_Commissioning.fbPart102Groups.aActivateButton[19] = FALSE, input disabled if: DALI_Commissioning.fbPart102Groups.aActivateButton[19] = FALSE
            OnMouseClick: execute { DALI_Commissioning.fbPart102Groups.aButtonClick[19] := TRUE; }
        Textfield (275,120 50x30), "20", colour toggle: DALI_Commissioning.fbPart102Groups.aShowAlarmState[20] = TRUE, invisible if: DALI_Commissioning.fbPart102Groups.aActivateButton[20] = FALSE, input disabled if: DALI_Commissioning.fbPart102Groups.aActivateButton[20] = FALSE
            OnMouseClick: execute { DALI_Commissioning.fbPart102Groups.aButtonClick[20] := TRUE; }
        Textfield (340,120 50x30), "21", colour toggle: DALI_Commissioning.fbPart102Groups.aShowAlarmState[21] = TRUE, invisible if: DALI_Commissioning.fbPart102Groups.aActivateButton[21] = FALSE, input disabled if: DALI_Commissioning.fbPart102Groups.aActivateButton[21] = FALSE
            OnMouseClick: execute { DALI_Commissioning.fbPart102Groups.aButtonClick[21] := TRUE; }
        Textfield (405,120 50x30), "22", colour toggle: DALI_Commissioning.fbPart102Groups.aShowAlarmState[22] = TRUE, invisible if: DALI_Commissioning.fbPart102Groups.aActivateButton[22] = FALSE, input disabled if: DALI_Commissioning.fbPart102Groups.aActivateButton[22] = FALSE
            OnMouseClick: execute { DALI_Commissioning.fbPart102Groups.aButtonClick[22] := TRUE; }
        Textfield (470,120 50x30), "23", colour toggle: DALI_Commissioning.fbPart102Groups.aShowAlarmState[23] = TRUE, invisible if: DALI_Commissioning.fbPart102Groups.aActivateButton[23] = FALSE, input disabled if: DALI_Commissioning.fbPart102Groups.aActivateButton[23] = FALSE
            OnMouseClick: execute { DALI_Commissioning.fbPart102Groups.aButtonClick[23] := TRUE; }
        Textfield (15,165 50x30), "24", colour toggle: DALI_Commissioning.fbPart102Groups.aShowAlarmState[24] = TRUE, invisible if: DALI_Commissioning.fbPart102Groups.aDeviceGroupState[24] = 0, input disabled if: DALI_Commissioning.fbPart102Groups.aDeviceGroupState[24] = 0
            OnMouseClick: execute { DALI_Commissioning.fbPart102Groups.aButtonClick[24] := TRUE; }
        Textfield (80,165 50x30), "25", colour toggle: DALI_Commissioning.fbPart102Groups.aShowAlarmState[25] = TRUE, invisible if: DALI_Commissioning.fbPart102Groups.aActivateButton[25] = FALSE, input disabled if: DALI_Commissioning.fbPart102Groups.aActivateButton[25] = FALSE
            OnMouseClick: execute { DALI_Commissioning.fbPart102Groups.aButtonClick[25] := TRUE; }
        Textfield (145,165 50x30), "26", colour toggle: DALI_Commissioning.fbPart102Groups.aShowAlarmState[26] = TRUE, invisible if: DALI_Commissioning.fbPart102Groups.aActivateButton[26] = FALSE, input disabled if: DALI_Commissioning.fbPart102Groups.aActivateButton[26] = FALSE
            OnMouseClick: execute { DALI_Commissioning.fbPart102Groups.aButtonClick[26] := TRUE; }
        Textfield (210,165 50x30), "27", colour toggle: DALI_Commissioning.fbPart102Groups.aShowAlarmState[27] = TRUE, invisible if: DALI_Commissioning.fbPart102Groups.aActivateButton[27] = FALSE, input disabled if: DALI_Commissioning.fbPart102Groups.aActivateButton[27] = FALSE
            OnMouseClick: execute { DALI_Commissioning.fbPart102Groups.aButtonClick[27] := TRUE; }
        Textfield (275,165 50x30), "28", colour toggle: DALI_Commissioning.fbPart102Groups.aShowAlarmState[28] = TRUE, invisible if: DALI_Commissioning.fbPart102Groups.aActivateButton[28] = FALSE, input disabled if: DALI_Commissioning.fbPart102Groups.aActivateButton[28] = FALSE
            OnMouseClick: execute { DALI_Commissioning.fbPart102Groups.aButtonClick[28] := TRUE; }
        Textfield (340,165 50x30), "29", colour toggle: DALI_Commissioning.fbPart102Groups.aShowAlarmState[29] = TRUE, invisible if: DALI_Commissioning.fbPart102Groups.aActivateButton[29] = FALSE, input disabled if: DALI_Commissioning.fbPart102Groups.aActivateButton[29] = FALSE
            OnMouseClick: execute { DALI_Commissioning.fbPart102Groups.aButtonClick[29] := TRUE; }
        Textfield (405,165 50x30), "30", colour toggle: DALI_Commissioning.fbPart102Groups.aShowAlarmState[30] = TRUE, invisible if: DALI_Commissioning.fbPart102Groups.aActivateButton[30] = FALSE, input disabled if: DALI_Commissioning.fbPart102Groups.aActivateButton[30] = FALSE
            OnMouseClick: execute { DALI_Commissioning.fbPart102Groups.aButtonClick[30] := TRUE; }
        Textfield (470,165 50x30), "31", colour toggle: DALI_Commissioning.fbPart102Groups.aShowAlarmState[31] = TRUE, invisible if: DALI_Commissioning.fbPart102Groups.aActivateButton[31] = FALSE, input disabled if: DALI_Commissioning.fbPart102Groups.aActivateButton[31] = FALSE
            OnMouseClick: execute { DALI_Commissioning.fbPart102Groups.aButtonClick[31] := TRUE; }
        Textfield (15,210 50x30), "32", colour toggle: DALI_Commissioning.fbPart102Groups.aShowAlarmState[32] = TRUE, invisible if: DALI_Commissioning.fbPart102Groups.aActivateButton[32] = FALSE, input disabled if: DALI_Commissioning.fbPart102Groups.aActivateButton[32] = FALSE
            OnMouseClick: execute { DALI_Commissioning.fbPart102Groups.aButtonClick[32] := TRUE; }
        Textfield (80,210 50x30), "33", colour toggle: DALI_Commissioning.fbPart102Groups.aShowAlarmState[33] = TRUE, invisible if: DALI_Commissioning.fbPart102Groups.aActivateButton[33] = FALSE, input disabled if: DALI_Commissioning.fbPart102Groups.aActivateButton[33] = FALSE
            OnMouseClick: execute { DALI_Commissioning.fbPart102Groups.aButtonClick[33] := TRUE; }
        Textfield (145,210 50x30), "34", colour toggle: DALI_Commissioning.fbPart102Groups.aShowAlarmState[34] = TRUE, invisible if: DALI_Commissioning.fbPart102Groups.aActivateButton[34] = FALSE, input disabled if: DALI_Commissioning.fbPart102Groups.aActivateButton[34] = FALSE
            OnMouseClick: execute { DALI_Commissioning.fbPart102Groups.aButtonClick[34] := TRUE; }
        Textfield (210,210 50x30), "35", colour toggle: DALI_Commissioning.fbPart102Groups.aShowAlarmState[35] = TRUE, invisible if: DALI_Commissioning.fbPart102Groups.aActivateButton[35] = FALSE, input disabled if: DALI_Commissioning.fbPart102Groups.aActivateButton[35] = FALSE
            OnMouseClick: execute { DALI_Commissioning.fbPart102Groups.aButtonClick[35] := TRUE; }
        Textfield (275,210 50x30), "36", colour toggle: DALI_Commissioning.fbPart102Groups.aShowAlarmState[36] = TRUE, invisible if: DALI_Commissioning.fbPart102Groups.aActivateButton[36] = FALSE, input disabled if: DALI_Commissioning.fbPart102Groups.aActivateButton[36] = FALSE
            OnMouseClick: execute { DALI_Commissioning.fbPart102Groups.aButtonClick[36] := TRUE; }
        Textfield (340,210 50x30), "37", colour toggle: DALI_Commissioning.fbPart102Groups.aShowAlarmState[37] = TRUE, invisible if: DALI_Commissioning.fbPart102Groups.aActivateButton[37] = FALSE, input disabled if: DALI_Commissioning.fbPart102Groups.aActivateButton[37] = FALSE
            OnMouseClick: execute { DALI_Commissioning.fbPart102Groups.aButtonClick[37] := TRUE; }
        Textfield (405,210 50x30), "38", colour toggle: DALI_Commissioning.fbPart102Groups.aShowAlarmState[38] = TRUE, invisible if: DALI_Commissioning.fbPart102Groups.aActivateButton[38] = FALSE, input disabled if: DALI_Commissioning.fbPart102Groups.aActivateButton[38] = FALSE
            OnMouseClick: execute { DALI_Commissioning.fbPart102Groups.aButtonClick[38] := TRUE; }
        Textfield (470,210 50x30), "39", colour toggle: DALI_Commissioning.fbPart102Groups.aShowAlarmState[39] = TRUE, invisible if: DALI_Commissioning.fbPart102Groups.aActivateButton[39] = FALSE, input disabled if: DALI_Commissioning.fbPart102Groups.aActivateButton[39] = FALSE
            OnMouseClick: execute { DALI_Commissioning.fbPart102Groups.aButtonClick[39] := TRUE; }
        Textfield (15,255 50x30), "40", colour toggle: DALI_Commissioning.fbPart102Groups.aShowAlarmState[40] = TRUE, invisible if: DALI_Commissioning.fbPart102Groups.aActivateButton[40] = FALSE, input disabled if: DALI_Commissioning.fbPart102Groups.aActivateButton[40] = FALSE
            OnMouseClick: execute { DALI_Commissioning.fbPart102Groups.aButtonClick[40] := TRUE; }
        Textfield (80,255 50x30), "41", colour toggle: DALI_Commissioning.fbPart102Groups.aShowAlarmState[41] = TRUE, invisible if: DALI_Commissioning.fbPart102Groups.aActivateButton[41] = FALSE, input disabled if: DALI_Commissioning.fbPart102Groups.aActivateButton[41] = FALSE
            OnMouseClick: execute { DALI_Commissioning.fbPart102Groups.aButtonClick[41] := TRUE; }
        Textfield (145,255 50x30), "42", colour toggle: DALI_Commissioning.fbPart102Groups.aShowAlarmState[42] = TRUE, invisible if: DALI_Commissioning.fbPart102Groups.aActivateButton[42] = FALSE, input disabled if: DALI_Commissioning.fbPart102Groups.aActivateButton[42] = FALSE
            OnMouseClick: execute { DALI_Commissioning.fbPart102Groups.aButtonClick[42] := TRUE; }
        Textfield (210,255 50x30), "43", colour toggle: DALI_Commissioning.fbPart102Groups.aShowAlarmState[43] = TRUE, invisible if: DALI_Commissioning.fbPart102Groups.aActivateButton[43] = FALSE, input disabled if: DALI_Commissioning.fbPart102Groups.aActivateButton[43] = FALSE
            OnMouseClick: execute { DALI_Commissioning.fbPart102Groups.aButtonClick[43] := TRUE; }
        Textfield (275,255 50x30), "44", colour toggle: DALI_Commissioning.fbPart102Groups.aShowAlarmState[44] = TRUE, invisible if: DALI_Commissioning.fbPart102Groups.aActivateButton[44] = FALSE, input disabled if: DALI_Commissioning.fbPart102Groups.aActivateButton[44] = FALSE
            OnMouseClick: execute { DALI_Commissioning.fbPart102Groups.aButtonClick[44] := TRUE; }
        Textfield (340,255 50x30), "45", colour toggle: DALI_Commissioning.fbPart102Groups.aShowAlarmState[45] = TRUE, invisible if: DALI_Commissioning.fbPart102Groups.aActivateButton[45] = FALSE, input disabled if: DALI_Commissioning.fbPart102Groups.aActivateButton[45] = FALSE
            OnMouseClick: execute { DALI_Commissioning.fbPart102Groups.aButtonClick[45] := TRUE; }
        Textfield (405,255 50x30), "46", colour toggle: DALI_Commissioning.fbPart102Groups.aShowAlarmState[46] = TRUE, invisible if: DALI_Commissioning.fbPart102Groups.aActivateButton[46] = FALSE, input disabled if: DALI_Commissioning.fbPart102Groups.aActivateButton[46] = FALSE
            OnMouseClick: execute { DALI_Commissioning.fbPart102Groups.aButtonClick[46] := TRUE; }
        Textfield (470,255 50x30), "47", colour toggle: DALI_Commissioning.fbPart102Groups.aShowAlarmState[47] = TRUE, invisible if: DALI_Commissioning.fbPart102Groups.aActivateButton[47] = FALSE, input disabled if: DALI_Commissioning.fbPart102Groups.aActivateButton[47] = FALSE
            OnMouseClick: execute { DALI_Commissioning.fbPart102Groups.aButtonClick[47] := TRUE; }
        Textfield (15,300 50x30), "48", colour toggle: DALI_Commissioning.fbPart102Groups.aShowAlarmState[48] = TRUE, invisible if: DALI_Commissioning.fbPart102Groups.aActivateButton[48] = FALSE, input disabled if: DALI_Commissioning.fbPart102Groups.aActivateButton[48] = FALSE
            OnMouseClick: execute { DALI_Commissioning.fbPart102Groups.aButtonClick[48] := TRUE; }
        Textfield (80,300 50x30), "49", colour toggle: DALI_Commissioning.fbPart102Groups.aShowAlarmState[49] = TRUE, invisible if: DALI_Commissioning.fbPart102Groups.aActivateButton[49] = FALSE, input disabled if: DALI_Commissioning.fbPart102Groups.aActivateButton[49] = FALSE
            OnMouseClick: execute { DALI_Commissioning.fbPart102Groups.aButtonClick[49] := TRUE; }
        Textfield (145,300 50x30), "50", colour toggle: DALI_Commissioning.fbPart102Groups.aShowAlarmState[50] = TRUE, invisible if: DALI_Commissioning.fbPart102Groups.aActivateButton[50] = FALSE, input disabled if: DALI_Commissioning.fbPart102Groups.aActivateButton[50] = FALSE
            OnMouseClick: execute { DALI_Commissioning.fbPart102Groups.aButtonClick[50] := TRUE; }
        Textfield (210,300 50x30), "51", colour toggle: DALI_Commissioning.fbPart102Groups.aShowAlarmState[51] = TRUE, invisible if: DALI_Commissioning.fbPart102Groups.aActivateButton[51] = FALSE, input disabled if: DALI_Commissioning.fbPart102Groups.aActivateButton[51] = FALSE
            OnMouseClick: execute { DALI_Commissioning.fbPart102Groups.aButtonClick[51] := TRUE; }
        Textfield (275,300 50x30), "52", colour toggle: DALI_Commissioning.fbPart102Groups.aShowAlarmState[52] = TRUE, invisible if: DALI_Commissioning.fbPart102Groups.aActivateButton[52] = FALSE, input disabled if: DALI_Commissioning.fbPart102Groups.aActivateButton[52] = FALSE
            OnMouseClick: execute { DALI_Commissioning.fbPart102Groups.aButtonClick[52] := TRUE; }
        Textfield (340,300 50x30), "53", colour toggle: DALI_Commissioning.fbPart102Groups.aShowAlarmState[53] = TRUE, invisible if: DALI_Commissioning.fbPart102Groups.aActivateButton[53] = FALSE, input disabled if: DALI_Commissioning.fbPart102Groups.aActivateButton[53] = FALSE
            OnMouseClick: execute { DALI_Commissioning.fbPart102Groups.aButtonClick[53] := TRUE; }
        Textfield (405,300 50x30), "54", colour toggle: DALI_Commissioning.fbPart102Groups.aShowAlarmState[54] = TRUE, invisible if: DALI_Commissioning.fbPart102Groups.aActivateButton[54] = FALSE, input disabled if: DALI_Commissioning.fbPart102Groups.aActivateButton[54] = FALSE
            OnMouseClick: execute { DALI_Commissioning.fbPart102Groups.aButtonClick[54] := TRUE; }
        Textfield (470,300 50x30), "55", colour toggle: DALI_Commissioning.fbPart102Groups.aShowAlarmState[55] = TRUE, invisible if: DALI_Commissioning.fbPart102Groups.aActivateButton[55] = FALSE, input disabled if: DALI_Commissioning.fbPart102Groups.aActivateButton[55] = FALSE
            OnMouseClick: execute { DALI_Commissioning.fbPart102Groups.aButtonClick[55] := TRUE; }
        Textfield (15,345 50x30), "56", colour toggle: DALI_Commissioning.fbPart102Groups.aShowAlarmState[56] = TRUE, invisible if: DALI_Commissioning.fbPart102Groups.aActivateButton[56] = FALSE, input disabled if: DALI_Commissioning.fbPart102Groups.aActivateButton[56] = FALSE
            OnMouseClick: execute { DALI_Commissioning.fbPart102Groups.aButtonClick[56] := TRUE; }
        Textfield (80,345 50x30), "57", colour toggle: DALI_Commissioning.fbPart102Groups.aShowAlarmState[57] = TRUE, invisible if: DALI_Commissioning.fbPart102Groups.aActivateButton[57] = FALSE, input disabled if: DALI_Commissioning.fbPart102Groups.aActivateButton[57] = FALSE
            OnMouseClick: execute { DALI_Commissioning.fbPart102Groups.aButtonClick[56] := TRUE; }
        Textfield (145,345 50x30), "58", colour toggle: DALI_Commissioning.fbPart102Groups.aShowAlarmState[58] = TRUE, invisible if: DALI_Commissioning.fbPart102Groups.aActivateButton[58] = FALSE, input disabled if: DALI_Commissioning.fbPart102Groups.aActivateButton[58] = FALSE
            OnMouseClick: execute { DALI_Commissioning.fbPart102Groups.aButtonClick[58] := TRUE; }
        Textfield (210,345 50x30), "59", colour toggle: DALI_Commissioning.fbPart102Groups.aShowAlarmState[59] = TRUE, invisible if: DALI_Commissioning.fbPart102Groups.aActivateButton[59] = FALSE, input disabled if: DALI_Commissioning.fbPart102Groups.aActivateButton[59] = FALSE
            OnMouseClick: execute { DALI_Commissioning.fbPart102Groups.aButtonClick[59] := TRUE; }
        Textfield (275,345 50x30), "60", colour toggle: DALI_Commissioning.fbPart102Groups.aShowAlarmState[60] = TRUE, invisible if: DALI_Commissioning.fbPart102Groups.aActivateButton[60] = FALSE, input disabled if: DALI_Commissioning.fbPart102Groups.aActivateButton[60] = FALSE
            OnMouseClick: execute { DALI_Commissioning.fbPart102Groups.aButtonClick[60] := TRUE; }
        Textfield (340,345 50x30), "61", colour toggle: DALI_Commissioning.fbPart102Groups.aShowAlarmState[61] = TRUE, invisible if: DALI_Commissioning.fbPart102Groups.aActivateButton[61] = FALSE, input disabled if: DALI_Commissioning.fbPart102Groups.aActivateButton[61] = FALSE
            OnMouseClick: execute { DALI_Commissioning.fbPart102Groups.aButtonClick[61] := TRUE; }
        Textfield (405,345 50x30), "62", colour toggle: DALI_Commissioning.fbPart102Groups.aShowAlarmState[62] = TRUE, invisible if: DALI_Commissioning.fbPart102Groups.aActivateButton[62] = FALSE, input disabled if: DALI_Commissioning.fbPart102Groups.aActivateButton[62] = FALSE
            OnMouseClick: execute { DALI_Commissioning.fbPart102Groups.aButtonClick[62] := TRUE; }
        Textfield (470,345 50x30), "63", colour toggle: DALI_Commissioning.fbPart102Groups.aShowAlarmState[63] = TRUE, invisible if: DALI_Commissioning.fbPart102Groups.aActivateButton[63] = FALSE, input disabled if: DALI_Commissioning.fbPart102Groups.aActivateButton[63] = FALSE
            OnMouseClick: execute { DALI_Commissioning.fbPart102Groups.aButtonClick[63] := TRUE; }
        WaitingSymbolFlower (230,170 70x70), invisible if: DALI_Commissioning.fbPart102Groups.bHideWaitSymbol
    Button (610,400 150x40), "Read"
        OnMouseClick: execute { DALI_Commissioning.fbPart102Groups.bRead := TRUE; }
    Button (610,450 150x40), "Write"
        OnMouseClick: execute { DALI_Commissioning.fbPart102Groups.bWrite := TRUE; }
    Button (610,100 150x40), "Switch On"
        OnMouseClick: execute { DALI_Commissioning.fbPart102Groups.bSwitchOn := TRUE; }
    Button (610,150 150x40), "Switch Off"
        OnMouseClick: execute { DALI_Commissioning.fbPart102Groups.bSwitchOff := TRUE; }
    Group (320,5 210x40)
        Textfield (0,0 120x40), "Choose group:"
        Button (130,0 80x40), "%s", text variable: DALI_Commissioning.fbPart102Groups.nGroupAddress
            OnMouseClick: write the text variable via Default, min 0, max 15, title "Choose group"
    Group (10,5 170x40)
        Textfield (0,0 110x40), "DALI Line:"
        Button (90,0 80x40), "%d", text variable: GVL_Internal.nDALILine
            OnMouseClick: write the text variable via Default, min 1, max 10, title "Choose line"
END_VISUALIZATION

// ---- POUs/DALI/DALI_Setup/VISUs/Visu_DALICommissioning/Visu_Part102Scenes.TcVIS
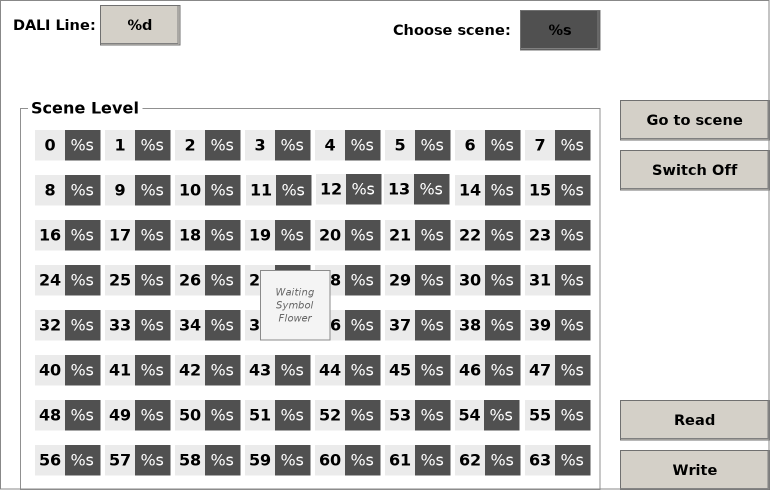
VISUALIZATION Visu_Part102Scenes  // 770x490
    GroupBox (20,100 580x390), "Scene Level"
        Group (85,30 65x30)
            Textfield (0,0 30x30), "1"
            Textfield (30,0 35x30), "%s", text variable: DALI_Commissioning.fbPart102Scenes.aScene[1], input disabled if: DALI_Commissioning.fbPart102Scenes.aNoShortAddress[1]
                p55702900: DALI_Commissioning.fbPart102Scenes.aFont[1]
                OnMouseClick: write the text variable via Default, min 0, max 255, title "Scene Value"
        Group (505,30 65x30)
            Textfield (0,0 30x30), "7"
            Textfield (30,0 35x30), "%s", text variable: DALI_Commissioning.fbPart102Scenes.aScene[7], input disabled if: DALI_Commissioning.fbPart102Scenes.aNoShortAddress[7]
                p55702900: DALI_Commissioning.fbPart102Scenes.aFont[7]
                OnMouseClick: write the text variable via Default, min 0, max 255, title "Scene Value"
        Group (435,30 65x30)
            Textfield (0,0 30x30), "6"
            Textfield (30,0 35x30), "%s", text variable: DALI_Commissioning.fbPart102Scenes.aScene[6], input disabled if: DALI_Commissioning.fbPart102Scenes.aNoShortAddress[6]
                p55702900: DALI_Commissioning.fbPart102Scenes.aFont[6]
                OnMouseClick: write the text variable via Default, min 0, max 255, title "Scene Value"
        Group (365,30 65x30)
            Textfield (0,0 30x30), "5"
            Textfield (30,0 35x30), "%s", text variable: DALI_Commissioning.fbPart102Scenes.aScene[5], input disabled if: DALI_Commissioning.fbPart102Scenes.aNoShortAddress[5]
                p55702900: DALI_Commissioning.fbPart102Scenes.aFont[5]
                OnMouseClick: write the text variable via Default, min 0, max 255, title "Scene Value"
        Group (295,30 65x30)
            Textfield (0,0 30x30), "4"
            Textfield (30,0 35x30), "%s", text variable: DALI_Commissioning.fbPart102Scenes.aScene[4], input disabled if: DALI_Commissioning.fbPart102Scenes.aNoShortAddress[4]
                p55702900: DALI_Commissioning.fbPart102Scenes.aFont[4]
                OnMouseClick: write the text variable via Default, min 0, max 255, title "Scene Value"
        Group (225,30 65x30)
            Textfield (0,0 30x30), "3"
            Textfield (30,0 35x30), "%s", text variable: DALI_Commissioning.fbPart102Scenes.aScene[3], input disabled if: DALI_Commissioning.fbPart102Scenes.aNoShortAddress[3]
                p55702900: DALI_Commissioning.fbPart102Scenes.aFont[3]
                OnMouseClick: write the text variable via Default, min 0, max 255, title "Scene Value"
        Group (155,30 65x30)
            Textfield (0,0 30x30), "2"
            Textfield (30,0 35x30), "%s", text variable: DALI_Commissioning.fbPart102Scenes.aScene[2], input disabled if: DALI_Commissioning.fbPart102Scenes.aNoShortAddress[2]
                p55702900: DALI_Commissioning.fbPart102Scenes.aFont[2]
                OnMouseClick: write the text variable via Default, min 0, max 255, title "Scene Value"
        Group (15,75 65x30)
            Textfield (0,0 30x30), "8"
            Textfield (30,0 35x30), "%s", text variable: DALI_Commissioning.fbPart102Scenes.aScene[8], input disabled if: DALI_Commissioning.fbPart102Scenes.aNoShortAddress[8]
                p55702900: DALI_Commissioning.fbPart102Scenes.aFont[8]
                OnMouseClick: write the text variable via Default, min 0, max 255, title "Scene Value"
        Group (15,120 65x30)
            Textfield (0,0 30x30), "16"
            Textfield (30,0 35x30), "%s", text variable: DALI_Commissioning.fbPart102Scenes.aScene[16], input disabled if: DALI_Commissioning.fbPart102Scenes.aNoShortAddress[16]
                p55702900: DALI_Commissioning.fbPart102Scenes.aFont[16]
                OnMouseClick: write the text variable via Default, min 0, max 255, title "Scene Value"
        Group (15,165 65x30)
            Textfield (0,0 30x30), "24"
            Textfield (30,0 35x30), "%s", text variable: DALI_Commissioning.fbPart102Scenes.aScene[24], input disabled if: DALI_Commissioning.fbPart102Scenes.aNoShortAddress[24]
                p55702900: DALI_Commissioning.fbPart102Scenes.aFont[24]
                OnMouseClick: write the text variable via Default, min 0, max 255, title "Scene Value"
        Group (15,210 65x30)
            Textfield (0,0 30x30), "32"
            Textfield (30,0 35x30), "%s", text variable: DALI_Commissioning.fbPart102Scenes.aScene[32], input disabled if: DALI_Commissioning.fbPart102Scenes.aNoShortAddress[32]
                p55702900: DALI_Commissioning.fbPart102Scenes.aFont[32]
                OnMouseClick: write the text variable via Default, min 0, max 255, title "Scene Value"
        Group (15,255 65x30)
            Textfield (0,0 30x30), "40"
            Textfield (30,0 35x30), "%s", text variable: DALI_Commissioning.fbPart102Scenes.aScene[40], input disabled if: DALI_Commissioning.fbPart102Scenes.aNoShortAddress[40]
                p55702900: DALI_Commissioning.fbPart102Scenes.aFont[40]
                OnMouseClick: write the text variable via Default, min 0, max 255, title "Scene Value"
        Group (15,300 65x30)
            Textfield (0,0 30x30), "48"
            Textfield (30,0 35x30), "%s", text variable: DALI_Commissioning.fbPart102Scenes.aScene[48], input disabled if: DALI_Commissioning.fbPart102Scenes.aNoShortAddress[48]
                p55702900: DALI_Commissioning.fbPart102Scenes.aFont[48]
                OnMouseClick: write the text variable via Default, min 0, max 255, title "Scene Value"
        Group (15,345 65x30)
            Textfield (0,0 30x30), "56"
            Textfield (30,0 35x30), "%s", text variable: DALI_Commissioning.fbPart102Scenes.aScene[56], input disabled if: DALI_Commissioning.fbPart102Scenes.aNoShortAddress[56]
                p55702900: DALI_Commissioning.fbPart102Scenes.aFont[56]
                OnMouseClick: write the text variable via Default, min 0, max 255, title "Scene Value"
        Group (85,75 65x30)
            Textfield (0,0 30x30), "9"
            Textfield (30,0 35x30), "%s", text variable: DALI_Commissioning.fbPart102Scenes.aScene[9], input disabled if: DALI_Commissioning.fbPart102Scenes.aNoShortAddress[9]
                p55702900: DALI_Commissioning.fbPart102Scenes.aFont[9]
                OnMouseClick: write the text variable via Default, min 0, max 255, title "Scene Value"
        Group (155,75 65x30)
            Textfield (0,0 30x30), "10"
            Textfield (30,0 35x30), "%s", text variable: DALI_Commissioning.fbPart102Scenes.aScene[10], input disabled if: DALI_Commissioning.fbPart102Scenes.aNoShortAddress[10]
                p55702900: DALI_Commissioning.fbPart102Scenes.aFont[10]
                OnMouseClick: write the text variable via Default, min 0, max 255, title "Scene Value"
        Group (226,75 65x30)
            Textfield (0,0 30x30), "11"
            Textfield (30,0 35x30), "%s", text variable: DALI_Commissioning.fbPart102Scenes.aScene[11], input disabled if: DALI_Commissioning.fbPart102Scenes.aNoShortAddress[11]
                p55702900: DALI_Commissioning.fbPart102Scenes.aFont[11]
                OnMouseClick: write the text variable via Default, min 0, max 255, title "Scene Value"
        Group (296,74 65x30)
            Textfield (0,0 30x30), "12"
            Textfield (30,0 35x30), "%s", text variable: DALI_Commissioning.fbPart102Scenes.aScene[12], input disabled if: DALI_Commissioning.fbPart102Scenes.aNoShortAddress[12]
                p55702900: DALI_Commissioning.fbPart102Scenes.aFont[12]
                OnMouseClick: write the text variable via Default, min 0, max 255, title "Scene Value"
        Group (364,74 65x30)
            Textfield (0,0 30x30), "13"
            Textfield (30,0 35x30), "%s", text variable: DALI_Commissioning.fbPart102Scenes.aScene[13], input disabled if: DALI_Commissioning.fbPart102Scenes.aNoShortAddress[13]
                p55702900: DALI_Commissioning.fbPart102Scenes.aFont[13]
                OnMouseClick: write the text variable via Default, min 0, max 255, title "Scene Value"
        Group (435,75 65x30)
            Textfield (0,0 30x30), "14"
            Textfield (30,0 35x30), "%s", text variable: DALI_Commissioning.fbPart102Scenes.aScene[14], input disabled if: DALI_Commissioning.fbPart102Scenes.aNoShortAddress[14]
                p55702900: DALI_Commissioning.fbPart102Scenes.aFont[14]
                OnMouseClick: write the text variable via Default, min 0, max 255, title "Scene Value"
        Group (505,75 65x30)
            Textfield (0,0 30x30), "15"
            Textfield (30,0 35x30), "%s", text variable: DALI_Commissioning.fbPart102Scenes.aScene[15], input disabled if: DALI_Commissioning.fbPart102Scenes.aNoShortAddress[15]
                p55702900: DALI_Commissioning.fbPart102Scenes.aFont[15]
                OnMouseClick: write the text variable via Default, min 0, max 255, title "Scene Value"
        Group (85,120 65x30)
            Textfield (0,0 30x30), "17"
            Textfield (30,0 35x30), "%s", text variable: DALI_Commissioning.fbPart102Scenes.aScene[17], input disabled if: DALI_Commissioning.fbPart102Scenes.aNoShortAddress[17]
                p55702900: DALI_Commissioning.fbPart102Scenes.aFont[17]
                OnMouseClick: write the text variable via Default, min 0, max 255, title "Scene Value"
        Group (155,120 65x30)
            Textfield (0,0 30x30), "18"
            Textfield (30,0 35x30), "%s", text variable: DALI_Commissioning.fbPart102Scenes.aScene[18], input disabled if: DALI_Commissioning.fbPart102Scenes.aNoShortAddress[18]
                p55702900: DALI_Commissioning.fbPart102Scenes.aFont[18]
                OnMouseClick: write the text variable via Default, min 0, max 255, title "Scene Value"
        Group (225,120 65x30)
            Textfield (0,0 30x30), "19"
            Textfield (30,0 35x30), "%s", text variable: DALI_Commissioning.fbPart102Scenes.aScene[19], input disabled if: DALI_Commissioning.fbPart102Scenes.aNoShortAddress[19]
                p55702900: DALI_Commissioning.fbPart102Scenes.aFont[19]
                OnMouseClick: write the text variable via Default, min 0, max 255, title "Scene Value"
        Group (295,120 65x30)
            Textfield (0,0 30x30), "20"
            Textfield (30,0 35x30), "%s", text variable: DALI_Commissioning.fbPart102Scenes.aScene[20], input disabled if: DALI_Commissioning.fbPart102Scenes.aNoShortAddress[20]
                p55702900: DALI_Commissioning.fbPart102Scenes.aFont[20]
                OnMouseClick: write the text variable via Default, min 0, max 255, title "Scene Value"
        Group (365,120 65x30)
            Textfield (0,0 30x30), "21"
            Textfield (30,0 35x30), "%s", text variable: DALI_Commissioning.fbPart102Scenes.aScene[21], input disabled if: DALI_Commissioning.fbPart102Scenes.aNoShortAddress[21]
                p55702900: DALI_Commissioning.fbPart102Scenes.aFont[21]
                OnMouseClick: write the text variable via Default, min 0, max 255, title "Scene Value"
        Group (435,120 65x30)
            Textfield (0,0 30x30), "22"
            Textfield (30,0 35x30), "%s", text variable: DALI_Commissioning.fbPart102Scenes.aScene[22], input disabled if: DALI_Commissioning.fbPart102Scenes.aNoShortAddress[22]
                p55702900: DALI_Commissioning.fbPart102Scenes.aFont[22]
                OnMouseClick: write the text variable via Default, min 0, max 255, title "Scene Value"
        Group (505,120 65x30)
            Textfield (0,0 30x30), "23"
            Textfield (30,0 35x30), "%s", text variable: DALI_Commissioning.fbPart102Scenes.aScene[23], input disabled if: DALI_Commissioning.fbPart102Scenes.aNoShortAddress[23]
                p55702900: DALI_Commissioning.fbPart102Scenes.aFont[23]
                OnMouseClick: write the text variable via Default, min 0, max 255, title "Scene Value"
        Group (85,165 65x30)
            Textfield (0,0 30x30), "25"
            Textfield (30,0 35x30), "%s", text variable: DALI_Commissioning.fbPart102Scenes.aScene[25], input disabled if: DALI_Commissioning.fbPart102Scenes.aNoShortAddress[25]
                p55702900: DALI_Commissioning.fbPart102Scenes.aFont[25]
                OnMouseClick: write the text variable via Default, min 0, max 255, title "Scene Value"
        Group (155,165 65x30)
            Textfield (0,0 30x30), "26"
            Textfield (30,0 35x30), "%s", text variable: DALI_Commissioning.fbPart102Scenes.aScene[26], input disabled if: DALI_Commissioning.fbPart102Scenes.aNoShortAddress[26]
                p55702900: DALI_Commissioning.fbPart102Scenes.aFont[26]
                OnMouseClick: write the text variable via Default, min 0, max 255, title "Scene Value"
        Group (225,165 65x30)
            Textfield (0,0 30x30), "27"
            Textfield (30,0 35x30), "%s", text variable: DALI_Commissioning.fbPart102Scenes.aScene[27], input disabled if: DALI_Commissioning.fbPart102Scenes.aNoShortAddress[27]
                p55702900: DALI_Commissioning.fbPart102Scenes.aFont[27]
                OnMouseClick: write the text variable via Default, min 0, max 255, title "Scene Value"
        Group (295,165 65x30)
            Textfield (0,0 30x30), "28"
            Textfield (30,0 35x30), "%s", text variable: DALI_Commissioning.fbPart102Scenes.aScene[28], input disabled if: DALI_Commissioning.fbPart102Scenes.aNoShortAddress[28]
                p55702900: DALI_Commissioning.fbPart102Scenes.aFont[28]
                OnMouseClick: write the text variable via Default, min 0, max 255, title "Scene Value"
        Group (365,165 65x30)
            Textfield (0,0 30x30), "29"
            Textfield (30,0 35x30), "%s", text variable: DALI_Commissioning.fbPart102Scenes.aScene[29], input disabled if: DALI_Commissioning.fbPart102Scenes.aNoShortAddress[29]
                p55702900: DALI_Commissioning.fbPart102Scenes.aFont[29]
                OnMouseClick: write the text variable via Default, min 0, max 255, title "Scene Value"
        Group (435,165 65x30)
            Textfield (0,0 30x30), "30"
            Textfield (30,0 35x30), "%s", text variable: DALI_Commissioning.fbPart102Scenes.aScene[30], input disabled if: DALI_Commissioning.fbPart102Scenes.aNoShortAddress[30]
                p55702900: DALI_Commissioning.fbPart102Scenes.aFont[30]
                OnMouseClick: write the text variable via Default, min 0, max 255, title "Scene Value"
        Group (505,165 65x30)
            Textfield (0,0 30x30), "31"
            Textfield (30,0 35x30), "%s", text variable: DALI_Commissioning.fbPart102Scenes.aScene[31], input disabled if: DALI_Commissioning.fbPart102Scenes.aNoShortAddress[31]
                p55702900: DALI_Commissioning.fbPart102Scenes.aFont[31]
                OnMouseClick: write the text variable via Default, min 0, max 255, title "Scene Value"
        Group (85,210 65x30)
            Textfield (0,0 30x30), "33"
            Textfield (30,0 35x30), "%s", text variable: DALI_Commissioning.fbPart102Scenes.aScene[33], input disabled if: DALI_Commissioning.fbPart102Scenes.aNoShortAddress[32]
                p55702900: DALI_Commissioning.fbPart102Scenes.aFont[33]
                OnMouseClick: write the text variable via Default, min 0, max 255, title "Scene Value"
        Group (155,210 65x30)
            Textfield (0,0 30x30), "34"
            Textfield (30,0 35x30), "%s", text variable: DALI_Commissioning.fbPart102Scenes.aScene[34], input disabled if: DALI_Commissioning.fbPart102Scenes.aNoShortAddress[34]
                p55702900: DALI_Commissioning.fbPart102Scenes.aFont[34]
                OnMouseClick: write the text variable via Default, min 0, max 255, title "Scene Value"
        Group (295,210 65x30)
            Textfield (0,0 30x30), "36"
            Textfield (30,0 35x30), "%s", text variable: DALI_Commissioning.fbPart102Scenes.aScene[36], input disabled if: DALI_Commissioning.fbPart102Scenes.aNoShortAddress[36]
                p55702900: DALI_Commissioning.fbPart102Scenes.aFont[36]
                OnMouseClick: write the text variable via Default, min 0, max 255
        Group (365,210 65x30)
            Textfield (0,0 30x30), "37"
            Textfield (30,0 35x30), "%s", text variable: DALI_Commissioning.fbPart102Scenes.aScene[37], input disabled if: DALI_Commissioning.fbPart102Scenes.aNoShortAddress[37]
                p55702900: DALI_Commissioning.fbPart102Scenes.aFont[37]
                OnMouseClick: write the text variable via Default, min 0, max 255, title "Scene Value"
        Group (435,210 65x30)
            Textfield (0,0 30x30), "38"
            Textfield (30,0 35x30), "%s", text variable: DALI_Commissioning.fbPart102Scenes.aScene[38], input disabled if: DALI_Commissioning.fbPart102Scenes.aNoShortAddress[38]
                p55702900: DALI_Commissioning.fbPart102Scenes.aFont[38]
                OnMouseClick: write the text variable via Default, min 0, max 255, title "Scene Value"
        Group (505,210 65x30)
            Textfield (0,0 30x30), "39"
            Textfield (30,0 35x30), "%s", text variable: DALI_Commissioning.fbPart102Scenes.aScene[39], input disabled if: DALI_Commissioning.fbPart102Scenes.aNoShortAddress[39]
                p55702900: DALI_Commissioning.fbPart102Scenes.aFont[39]
                OnMouseClick: write the text variable via Default, min 0, max 255, title "Scene Value"
        Group (85,255 65x30)
            Textfield (0,0 30x30), "41"
            Textfield (30,0 35x30), "%s", text variable: DALI_Commissioning.fbPart102Scenes.aScene[41], input disabled if: DALI_Commissioning.fbPart102Scenes.aNoShortAddress[41]
                p55702900: DALI_Commissioning.fbPart102Scenes.aFont[41]
                OnMouseClick: write the text variable via Default, min 0, max 255, title "Scene Value"
        Group (155,255 65x30)
            Textfield (0,0 30x30), "42"
            Textfield (30,0 35x30), "%s", text variable: DALI_Commissioning.fbPart102Scenes.aScene[42], input disabled if: DALI_Commissioning.fbPart102Scenes.aNoShortAddress[42]
                p55702900: DALI_Commissioning.fbPart102Scenes.aFont[42]
                OnMouseClick: write the text variable via Default, min 0, max 255, title "Scene Value"
        Group (225,210 65x30)
            Textfield (0,0 30x30), "35"
            Textfield (30,0 35x30), "%s", text variable: DALI_Commissioning.fbPart102Scenes.aScene[35], input disabled if: DALI_Commissioning.fbPart102Scenes.aNoShortAddress[35]
                p55702900: DALI_Commissioning.fbPart102Scenes.aFont[35]
                OnMouseClick: write the text variable via Default, min 0, max 255, title "Scene Value"
        Group (225,255 65x30)
            Textfield (0,0 30x30), "43"
            Textfield (30,0 35x30), "%s", text variable: DALI_Commissioning.fbPart102Scenes.aScene[43], input disabled if: DALI_Commissioning.fbPart102Scenes.aNoShortAddress[43]
                p55702900: DALI_Commissioning.fbPart102Scenes.aFont[43]
                OnMouseClick: write the text variable via Default, min 0, max 255, title "Scene Value"
        Group (295,255 65x30)
            Textfield (0,0 30x30), "44"
            Textfield (30,0 35x30), "%s", text variable: DALI_Commissioning.fbPart102Scenes.aScene[44], input disabled if: DALI_Commissioning.fbPart102Scenes.aNoShortAddress[44]
                p55702900: DALI_Commissioning.fbPart102Scenes.aFont[44]
                OnMouseClick: write the text variable via Default, min 0, max 255, title "Scene Value"
        Group (365,255 65x30)
            Textfield (0,0 30x30), "45"
            Textfield (30,0 35x30), "%s", text variable: DALI_Commissioning.fbPart102Scenes.aScene[45], input disabled if: DALI_Commissioning.fbPart102Scenes.aNoShortAddress[45]
                p55702900: DALI_Commissioning.fbPart102Scenes.aFont[45]
                OnMouseClick: write the text variable via Default, min 0, max 255, title "Scene Value"
        Group (435,255 65x30)
            Textfield (0,0 30x30), "46"
            Textfield (30,0 35x30), "%s", text variable: DALI_Commissioning.fbPart102Scenes.aScene[46], input disabled if: DALI_Commissioning.fbPart102Scenes.aNoShortAddress[46]
                p55702900: DALI_Commissioning.fbPart102Scenes.aFont[46]
                OnMouseClick: write the text variable via Default, min 0, max 255, title "Scene Value"
        Group (505,255 65x30)
            Textfield (0,0 30x30), "47"
            Textfield (30,0 35x30), "%s", text variable: DALI_Commissioning.fbPart102Scenes.aScene[47], input disabled if: DALI_Commissioning.fbPart102Scenes.aNoShortAddress[47]
                p55702900: DALI_Commissioning.fbPart102Scenes.aFont[47]
                OnMouseClick: write the text variable via Default, min 0, max 255, title "Scene Value"
        Group (85,300 65x30)
            Textfield (0,0 30x30), "49"
            Textfield (30,0 35x30), "%s", text variable: DALI_Commissioning.fbPart102Scenes.aScene[49], input disabled if: DALI_Commissioning.fbPart102Scenes.aNoShortAddress[49]
                p55702900: DALI_Commissioning.fbPart102Scenes.aFont[49]
                OnMouseClick: write the text variable via Default, min 0, max 255, title "Scene Value"
        Group (155,300 65x30)
            Textfield (0,0 30x30), "50"
            Textfield (30,0 35x30), "%s", text variable: DALI_Commissioning.fbPart102Scenes.aScene[50], input disabled if: DALI_Commissioning.fbPart102Scenes.aNoShortAddress[50]
                p55702900: DALI_Commissioning.fbPart102Scenes.aFont[50]
                OnMouseClick: write the text variable via Default, min 0, max 255, title "Scene Value"
        Group (225,300 65x30)
            Textfield (0,0 30x30), "51"
            Textfield (30,0 35x30), "%s", text variable: DALI_Commissioning.fbPart102Scenes.aScene[51], input disabled if: DALI_Commissioning.fbPart102Scenes.aNoShortAddress[51]
                p55702900: DALI_Commissioning.fbPart102Scenes.aFont[51]
                OnMouseClick: write the text variable via Default, min 0, max 255, title "Scene Value"
        Group (295,300 65x30)
            Textfield (0,0 30x30), "52"
            Textfield (30,0 35x30), "%s", text variable: DALI_Commissioning.fbPart102Scenes.aScene[52], input disabled if: DALI_Commissioning.fbPart102Scenes.aNoShortAddress[52]
                p55702900: DALI_Commissioning.fbPart102Scenes.aFont[52]
                OnMouseClick: write the text variable via Default, min 0, max 255, title "Scene Value"
        Group (365,300 65x30)
            Textfield (0,0 30x30), "53"
            Textfield (30,0 35x30), "%s", text variable: DALI_Commissioning.fbPart102Scenes.aScene[53], input disabled if: DALI_Commissioning.fbPart102Scenes.aNoShortAddress[53]
                p55702900: DALI_Commissioning.fbPart102Scenes.aFont[53]
                OnMouseClick: write the text variable via Default, min 0, max 255, title "Scene Value"
        Group (435,300 64x30)
            Textfield (0,0 29x30), "54"
            Textfield (29,0 35x30), "%s", text variable: DALI_Commissioning.fbPart102Scenes.aScene[54], input disabled if: DALI_Commissioning.fbPart102Scenes.aNoShortAddress[54]
                p55702900: DALI_Commissioning.fbPart102Scenes.aFont[54]
                OnMouseClick: write the text variable via Default, min 0, max 255, title "Scene Value"
        Group (505,300 65x30)
            Textfield (0,0 30x30), "55"
            Textfield (30,0 35x30), "%s", text variable: DALI_Commissioning.fbPart102Scenes.aScene[55], input disabled if: DALI_Commissioning.fbPart102Scenes.aNoShortAddress[55]
                p55702900: DALI_Commissioning.fbPart102Scenes.aFont[55]
                OnMouseClick: write the text variable via Default, min 0, max 255, title "Scene Value"
        Group (85,345 65x30)
            Textfield (0,0 30x30), "57"
            Textfield (30,0 35x30), "%s", text variable: DALI_Commissioning.fbPart102Scenes.aScene[57], input disabled if: DALI_Commissioning.fbPart102Scenes.aNoShortAddress[57]
                p55702900: DALI_Commissioning.fbPart102Scenes.aFont[57]
                OnMouseClick: write the text variable via Default, min 0, max 255, title "Scene Value"
        Group (155,345 65x30)
            Textfield (0,0 30x30), "58"
            Textfield (30,0 35x30), "%s", text variable: DALI_Commissioning.fbPart102Scenes.aScene[58], input disabled if: DALI_Commissioning.fbPart102Scenes.aNoShortAddress[58]
                p55702900: DALI_Commissioning.fbPart102Scenes.aFont[58]
                OnMouseClick: write the text variable via Default, min 0, max 255, title "Scene Value"
        Group (225,345 65x30)
            Textfield (0,0 30x30), "59"
            Textfield (30,0 35x30), "%s", text variable: DALI_Commissioning.fbPart102Scenes.aScene[59], input disabled if: DALI_Commissioning.fbPart102Scenes.aNoShortAddress[59]
                p55702900: DALI_Commissioning.fbPart102Scenes.aFont[59]
                OnMouseClick: write the text variable via Default, min 0, max 255, title "Scene Value"
        Group (295,345 65x30)
            Textfield (0,0 30x30), "60"
            Textfield (30,0 35x30), "%s", text variable: DALI_Commissioning.fbPart102Scenes.aScene[60], input disabled if: DALI_Commissioning.fbPart102Scenes.aNoShortAddress[60]
                p55702900: DALI_Commissioning.fbPart102Scenes.aFont[60]
                OnMouseClick: write the text variable via Default, min 0, max 255, title "Scene Value"
        Group (365,345 65x30)
            Textfield (0,0 30x30), "61"
            Textfield (30,0 35x30), "%s", text variable: DALI_Commissioning.fbPart102Scenes.aScene[61], input disabled if: DALI_Commissioning.fbPart102Scenes.aNoShortAddress[61]
                p55702900: DALI_Commissioning.fbPart102Scenes.aFont[61]
                OnMouseClick: write the text variable via Default, min 0, max 255, title "Scene Value"
        Group (435,345 65x30)
            Textfield (0,0 30x30), "62"
            Textfield (30,0 35x30), "%s", text variable: DALI_Commissioning.fbPart102Scenes.aScene[62], input disabled if: DALI_Commissioning.fbPart102Scenes.aNoShortAddress[62]
                p55702900: DALI_Commissioning.fbPart102Scenes.aFont[62]
                OnMouseClick: write the text variable via Default, min 0, max 255, title "Scene Value"
        Group (505,345 65x30)
            Textfield (0,0 30x30), "63"
            Textfield (30,0 35x30), "%s", text variable: DALI_Commissioning.fbPart102Scenes.aScene[63], input disabled if: DALI_Commissioning.fbPart102Scenes.aNoShortAddress[63]
                p55702900: DALI_Commissioning.fbPart102Scenes.aFont[63]
                OnMouseClick: write the text variable via Default, min 0, max 255, title "Scene Value"
        WaitingSymbolFlower (240,170 70x70), invisible if: DALI_Commissioning.fbPart102Scenes.bHideWaitSymbol
        Group (15,30 65x30)
            Textfield (0,0 30x30), "0"
            Textfield (30,0 35x30), "%s", text variable: DALI_Commissioning.fbPart102Scenes.aScene[0], input disabled if: DALI_Commissioning.fbPart102Scenes.aNoShortAddress[0]
                p55702900: DALI_Commissioning.fbPart102Scenes.aFont[0]
                OnMouseClick: write the text variable via Default, min 0, max 255, title "Scene Value"
    Button (620,400 150x40), "Read"
        OnMouseClick: execute { DALI_Commissioning.fbPart102Scenes.bRead := TRUE; }
    Button (620,450 150x40), "Write"
        OnMouseClick: execute { DALI_Commissioning.fbPart102Scenes.bWrite := TRUE; }
    Button (620,100 150x40), "Go to scene"
        OnMouseClick: execute { DALI_Commissioning.fbPart102Scenes.bGoToScene := TRUE; }
    Button (620,150 150x40), "Switch Off"
        OnMouseClick: execute { DALI_Commissioning.fbPart102Scenes.bSwitchOff := TRUE; }
    Textfield (390,10 120x40), "Choose scene:"
    Button (520,10 80x40), "%s", text variable: DALI_Commissioning.fbPart102Scenes.nScene
        OnMouseClick: write the text variable via Default, min 0, max 15, title "Choose scene"
    Group (10,5 170x40)
        Textfield (0,0 110x40), "DALI Line:"
        Button (90,0 80x40), "%d", text variable: GVL_Internal.nDALILine
            OnMouseClick: write the text variable via Default, min 1, max 10, title "Choose line"
END_VISUALIZATION

// ---- POUs/DALI/DALI_Setup/VISUs/Visu_DALICommissioning/Visu_Part103Identify.TcVIS
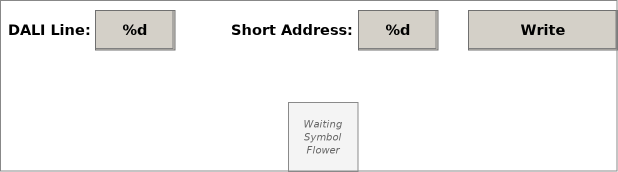
VISUALIZATION Visu_Part103Identify  // 618x172
    Button (468,10 150x40), "Write"
        OnMouseClick: execute { DALI_Commissioning.fbPart103IdentifyDevice.bWrite := TRUE; }
    WaitingSymbolFlower (288,102 70x70), invisible if: DALI_Commissioning.fbPart103MemoryPages.bHideWaitSymbol
    Textfield (228,10 130x40), "Short Address:"
    Button (358,10 80x40), "%d", text variable: DALI_Commissioning.fbPart103IdentifyDevice.nAddress
        OnMouseClick: write the text variable via Default, min 0, max 63, title "Insert Short Address"
    Group (5,10 170x40)
        Textfield (0,0 110x40), "DALI Line:"
        Button (90,0 80x40), "%d", text variable: GVL_Internal.nDALILine
            OnMouseClick: write the text variable via Default, min 1, max 10, title "Choose line"
END_VISUALIZATION

// ---- POUs/DALI/DALI_Setup/VISUs/Visu_DALICommissioning/Visu_Part205.TcVIS
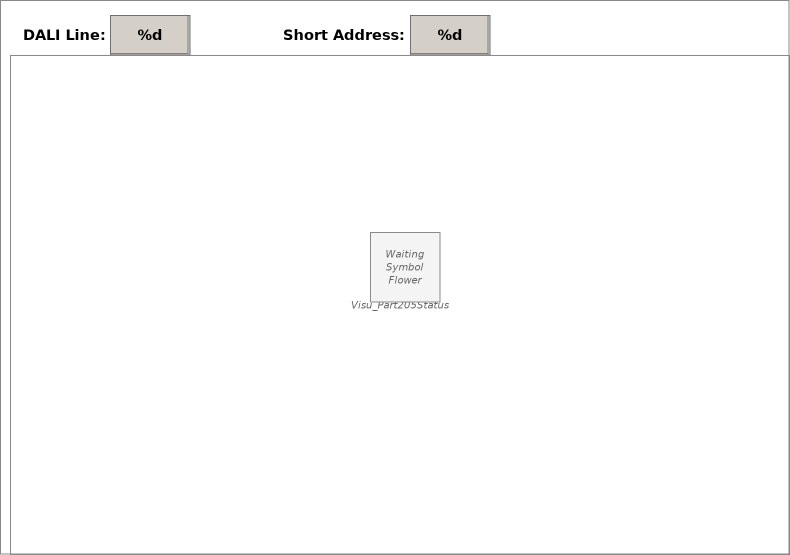
VISUALIZATION Visu_Part205  // 790x555
    Group (280,15 210x40)
        Textfield (0,0 130x40), "Short Address:"
        Button (130,0 80x40), "%d", text variable: DALI_Commissioning.fbPart205Incandescent.nAddress
            OnMouseClick: write the text variable via Default, min 0, max 63, title "Insert Short Address"
    Group (20,15 170x40)
        Textfield (0,0 110x40), "DALI Line:"
        Button (90,0 80x40), "%d", text variable: GVL_Internal.nDALILine
            OnMouseClick: write the text variable via Default, min 1, max 10, title "Choose line"
    TabControl (10,55 780x500)
        shows Visu_Part205Status()
        shows Visu_Part205Parameters()
        shows Visu_Part202Parameters()
        [0]: TabTitle=Status
        [1]: TabTitle=Parameters
        [2]: TabTitle=Parameters
    WaitingSymbolFlower (370,232 70x70), invisible if: DALI_Commissioning.fbPart205Incandescent.bHideWaitSymbol
END_VISUALIZATION

// ---- POUs/DALI/DALI_Setup/VISUs/Visu_DALICommissioning/Visu_Part300GenericDevice.TcVIS
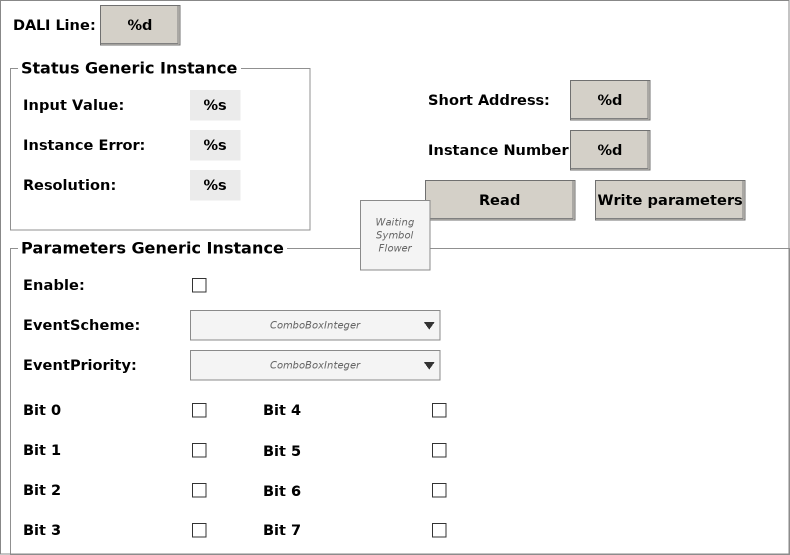
VISUALIZATION Visu_Part300GenericDevice  // 790x555
    GroupBox (10,240 780x315), "Parameters Generic Instance"
        Textfield (10,30 150x30), "Enable:"
        Checkbox (180,30 30x30), variable: DALI_Commissioning.fbPart300GenericDevice.bEnable
        Textfield (10,110 150x30), "EventPriority:"
        Textfield (10,195 100x30), "Bit 1"
        Textfield (10,155 100x30), "Bit 0"
        Checkbox (180,155 30x30), variable: DALI_Commissioning.fbPart300GenericDevice.bBit0
        Checkbox (180,195 30x30), variable: DALI_Commissioning.fbPart300GenericDevice.bBit1
        Textfield (10,235 100x30), "Bit 2"
        Textfield (250,155 100x30), "Bit 4"
        Textfield (250,196 100x30), "Bit 5"
        Checkbox (420,195 30x30), variable: DALI_Commissioning.fbPart300GenericDevice.bBit5
        Checkbox (420,155 30x30), variable: DALI_Commissioning.fbPart300GenericDevice.bBit4
        Checkbox (180,275 30x30), variable: DALI_Commissioning.fbPart300GenericDevice.bBit3
        Checkbox (180,235 30x30), variable: DALI_Commissioning.fbPart300GenericDevice.bBit2
        ComboBoxInteger (180,70 250x30), variable: DALI_Commissioning.fbPart300GenericDevice.eEventScheme, text list: 'EventScheme'
        Textfield (10,70 150x30), "EventScheme:"
        Textfield (250,236 100x30), "Bit 6"
        ComboBoxInteger (180,110 250x30), variable: DALI_Commissioning.fbPart300GenericDevice.eEventPriority, text list: 'EventPriority'
        Textfield (10,275 100x30), "Bit 3"
        Checkbox (420,235 30x30), variable: DALI_Commissioning.fbPart300GenericDevice.bBit6
        Checkbox (420,275 30x30), variable: DALI_Commissioning.fbPart300GenericDevice.bBit7
        Textfield (250,275 100x30), "Bit 7"
    GroupBox (10,60 300x170), "Status Generic Instance"
        Textfield (180,30 50x30), "%s", text variable: DALI_Commissioning.fbPart300GenericDevice.nInputValue
        Textfield (180,70 50x30), "%s", text variable: DALI_Commissioning.fbPart300GenericDevice.nInstanceError
        Textfield (180,110 50x30), "%s", text variable: DALI_Commissioning.fbPart300GenericDevice.nResolution
        Textfield (10,30 160x30), "Input Value:"
        Textfield (10,70 160x30), "Instance Error:"
        Textfield (10,110 160x30), "Resolution:"
    Button (425,180 150x40), "Read"
        OnMouseClick: execute { DALI_Commissioning.fbPart300GenericDevice.bRead := TRUE; }
    WaitingSymbolFlower (360,200 70x70), invisible if: DALI_Commissioning.fbPart300GenericDevice.bHideWaitSymbol
    Button (595,180 150x40), "Write parameters"
        OnMouseClick: execute { DALI_Commissioning.fbPart300GenericDevice.bWrite := TRUE; }
    Textfield (425,130 150x40), "Instance Number:"
    Textfield (425,80 150x40), "Short Address:"
    Button (570,80 80x40), "%d", text variable: DALI_Commissioning.fbPart300GenericDevice.nAddress
        OnMouseClick: write the text variable via Default, min 0, max 63, title "Insert Short Address"
    Button (570,130 80x40), "%d", text variable: DALI_Commissioning.fbPart300GenericDevice.nInstanceAddress
        OnMouseClick: write the text variable via Default, min 0, max 31, title "Insert instance number"
    Group (10,5 170x40)
        Textfield (0,0 110x40), "DALI Line:"
        Button (90,0 80x40), "%d", text variable: GVL_Internal.nDALILine
            OnMouseClick: write the text variable via Default, min 1, max 10, title "Choose line"
END_VISUALIZATION
